	fbDiagnosisEtherCATSlaveWc0				:ARRAY[E_EtherCATSlave.Drive14_AZD4A_KED..E_EtherCATSlave.Drive14_AZD4A_KED] OF FB_DiagnosisEtherCATSlaveWc0
																														(	E_EtherCATSlave.Drive14_AZD4A_KED
																															);	//EtherCAT Slave診断用FB
END_VAR

bError:=EtherCATMasterDiagnosis() OR EtherCATSlaveDiagnosis();

METHOD INTERNAL EtherCATMasterDiagnosis : BOOL
//EtherCATマスター診断
	//デバイス2
	fbDiagnosisEtherCATMaster2(	fbFrmWcStateDiagnosis	:=fbFrmWcStateDiagnosis2,
								fbFrmStateDiagnosis		:=fbFrmStateDiagnosis2);

	//デバイス6
	fbDiagnosisEtherCATMaster6(	fbFrmWcStateDiagnosis	:=fbFrmWcStateDiagnosis6,
								fbFrmStateDiagnosis		:=fbFrmStateDiagnosis6);

	//すべて問題なしで出力
	EtherCATMasterDiagnosis:= fbDiagnosisEtherCATMaster2.bError OR fbDiagnosisEtherCATMaster6.bError;
END_METHOD

METHOD INTERNAL EtherCATSlaveDiagnosis : BOOL
//EtherCATスレーブ診断
	fbDiagnosisEtherCATSlaveWc2[E_EtherCATSlave.Term12_EL2911]();
	fbDiagnosisEtherCATSlaveWc0[E_EtherCATSlave.Drive14_AZD4A_KED]();
	
	EtherCATSlaveDiagnosis:=fbDiagnosisEtherCATSlaveWc2[E_EtherCATSlave.Term12_EL2911].bError OR fbDiagnosisEtherCATSlaveWc0[E_EtherCATSlave.Drive14_AZD4A_KED].bError;

	FOR eEtherCATSlave := E_EtherCATSlave.Term2_EL9410 TO E_EtherCATSlave.Term11_EL1088 DO
		fbDiagnosisEtherCATSlaveWc1[eEtherCATSlave]();
		EtherCATSlaveDiagnosis:=EtherCATSlaveDiagnosis OR fbDiagnosisEtherCATSlaveWc1[eEtherCATSlave].bError;
	END_FOR
END_METHOD

END_FUNCTION_BLOCK

// ---- 01_Submodules/Diagnosis/EtherCAT Master/FB_FrmWcStateDiagnosis.TcPOU
FUNCTION_BLOCK FB_FrmWcStateDiagnosis
VAR_IN_OUT
	eEtherCATMaster				:E_EtherCATMaster;	
END_VAR
VAR_OUTPUT
	bError						:BOOL;								//エラー発生を出力
END_VAR
VAR
	uiFrmWcState 		AT%I*	:UINT;								//PDデータとリンク
	
	sMasterName					:STRING;
	
	bErrorState					:ARRAY[0..15] OF BOOL;				//各ステートエラー
	fbBitREdge					:ARRAY[0..15] OF R_TRIG;
	bSendMsgMem					:ARRAY[0..14] OF BOOL;				//メッセージ送信を記憶	
	sSendMsgString				:STRING;							//送信メッセージのアーギュメント用
	bSendMsg					:BOOL;								//メッセージ送信予約
	fbMessage					:ARRAY[0..1] OF FB_TcMessage;
	i							:INT;
END_VAR

//マスター名を入力
	IF sMasterName<>TO_STRING(eEtherCATMaster) THEN
		sMasterName:=TO_STRING(eEtherCATMaster);
	END_IF

//エラー状態を出力
	bError:= uiFrmWcState<>0 ;
	
//サイクリックフレームごとのワーキングカウンターチェック、エラーは複数発生する可能性があるので全bitチェック
	FOR i := 0 TO 15 DO
		bErrorState[i]:=(uiFrmWcState AND SHL(1,i))<>0;
	END_FOR
	
//結果をEventloggerへ
	bSendMsg:=FALSE;	//メッセージ送信予約をリセット

	FOR i := 0 TO 14 BY 1 DO
		//エラーの立ち上がりエッジを検出
		fbBitREdge[i](CLK:=bErrorState[i]);
		
		//まだ送信していなければ、送信用の文字列作成
		IF NOT bSendMsgMem[i] AND fbBitREdge[i].Q THEN
			
			sSendMsgString:=CONCAT(sSendMsgString, CONCAT(INT_TO_STRING(i+1), '. '));	//送信メッセージのアーギュメント作成

			bSendMsg:=TRUE;		//メッセージ送信予約をセット
			bSendMsgMem[i]:=TRUE;	//メッセージ送信を記憶
			
		END_IF
		
		//エラーがリセットされたらメッセージ送信気を記憶をリセット
		IF NOT bErrorState[i] THEN
			bSendMsgMem[i]:=FALSE;
		END_IF
		
	END_FOR
	
	IF bSendMsg THEN
		fbMessage[0].ipArguments.Clear().AddString(sSendMsgString).AddString(sMasterName);
		fbMessage[0].Send();
		
		bSendMsg:=FALSE;
		sSendMsgString:='';
	END_IF
	
	//全体判定用
	fbBitREdge[15](CLK:=bErrorState[15]);
	
	IF fbBitREdge[15].Q THEN
		fbMessage[1].ipArguments.Clear().AddString(sMasterName);
		fbMessage[1].Send();
	END_IF

//FB_Init は常に暗黙的に使用可能で、主に初期化に使用されます。
//戻り値は評価されません。特定の結果を得るために、メソッドを明示的に宣言し、
//そのメソッドに標準の初期化コードをもったコードを追加することができます。戻り値を評価できます。
METHOD FB_Init: BOOL
VAR_INPUT
    bInitRetains: BOOL; // TRUE: 保持変数は初期化されます (ウォーム リセット、あるいはコールド リセット)
    bInCopyCode: BOOL;  // TRUE: 後でコードをコピーする (オンライン変更) ために、インスタンスをコピーします。
END_VAR
fbMessage[0].CreateEx(TC_EVENTS.TkEtherCATMasterDiagnosisEventClass.WrongWorkingCounterEtherCATCommandReceived);
fbMessage[1].CreateEx(TC_EVENTS.TkEtherCATMasterDiagnosisEventClass.CompleteFrameMissing);
END_METHOD

END_FUNCTION_BLOCK

// ---- 01_Submodules/Diagnosis/EtherCAT Master/FB_FrmStateDiagnosis.TcPOU
FUNCTION_BLOCK FB_FrmStateDiagnosis
VAR_IN_OUT
	eEtherCATMaster				:E_EtherCATMaster;	
END_VAR
VAR_OUTPUT
	bError						:BOOL;								//エラー発生を出力
END_VAR
VAR
	uiFrmState 			AT%I*	:UINT;								//PDデータとリンク
	
	sMasterName					:STRING;
	
	bErrorState					:ARRAY[0..15] OF BOOL;				//各ステートエラー
	fbBitREdge					:ARRAY[0..15] OF R_TRIG;
	bSendMsgMem					:ARRAY[0..14] OF BOOL;				//メッセージ送信を記憶	
	sSendMsgString				:STRING;							//送信メッセージのアーギュメント用
	bSendMsg					:BOOL;								//メッセージ送信予約
	fbMessage					:ARRAY[0..1] OF FB_TcMessage;
	i							:INT;
END_VAR

//マスター名を入力
	IF sMasterName<>TO_STRING(eEtherCATMaster) THEN
		sMasterName:=TO_STRING(eEtherCATMaster);
	END_IF

//エラー状態を出力
	bError:= uiFrmState<>0 ;
	
//サイクリックフレームごとのワーキングカウンターチェック、エラーは複数発生する可能性があるので全bitチェック
	FOR i := 0 TO 15 DO
		bErrorState[i]:=(uiFrmState AND SHL(1,i))<>0;
	END_FOR
	
//結果をEventloggerへ
	bSendMsg:=FALSE;	//メッセージ送信予約をリセット

	FOR i := 0 TO 14 BY 1 DO
		//エラーの立ち上がりエッジを検出
		fbBitREdge[i](CLK:=bErrorState[i]);
		
		//まだ送信していなければ、送信用の文字列作成
		IF NOT bSendMsgMem[i] AND fbBitREdge[i].Q THEN
			
			sSendMsgString:=CONCAT(sSendMsgString, CONCAT(INT_TO_STRING(i+1), '. '));	//送信メッセージのアーギュメント作成

			bSendMsg:=TRUE;		//メッセージ送信予約をセット
			bSendMsgMem[i]:=TRUE;	//メッセージ送信を記憶
			
		END_IF
		
		//エラーがリセットされたらメッセージ送信気を記憶をリセット
		IF NOT bErrorState[i] THEN
			bSendMsgMem[i]:=FALSE;
		END_IF
		
	END_FOR
	
	IF bSendMsg THEN
		fbMessage[0].ipArguments.Clear().AddString(sSendMsgString).AddString(sMasterName);
		fbMessage[0].Send();
		
		bSendMsg:=FALSE;
		sSendMsgString:='';
	END_IF
	
	//全体判定用
	fbBitREdge[15](CLK:=bErrorState[15]);
	
	IF fbBitREdge[15].Q THEN
		fbMessage[1].ipArguments.Clear().AddString(sMasterName);
		fbMessage[1].Send();
	END_IF

//FB_Init は常に暗黙的に使用可能で、主に初期化に使用されます。
//戻り値は評価されません。特定の結果を得るために、メソッドを明示的に宣言し、
//そのメソッドに標準の初期化コードをもったコードを追加することができます。戻り値を評価できます。
METHOD FB_Init: BOOL
VAR_INPUT
    bInitRetains: BOOL; // TRUE: 保持変数は初期化されます (ウォーム リセット、あるいはコールド リセット)
    bInCopyCode: BOOL;  // TRUE: 後でコードをコピーする (オンライン変更) ために、インスタンスをコピーします。
END_VAR
fbMessage[0].CreateEx(TC_EVENTS.TkEtherCATMasterDiagnosisEventClass.EtherCATCommandNotSentNOPRequested);
fbMessage[1].CreateEx(TC_EVENTS.TkEtherCATMasterDiagnosisEventClass.CompleteFrameNotSent);
END_METHOD

END_FUNCTION_BLOCK

// ---- 01_Submodules/Diagnosis/EtherCAT Master/FB_DiagnosisEtherCATMaster.TcPOU
FUNCTION_BLOCK FB_DiagnosisEtherCATMaster
VAR_OUTPUT
	bError						:BOOL;								//エラー発生を出力
END_VAR
VAR_IN_OUT
	fbFrmWcStateDiagnosis		:ARRAY[*] OF FB_FrmWcStateDiagnosis;
	fbFrmStateDiagnosis			:ARRAY[*] OF FB_FrmStateDiagnosis;
END_VAR
VAR
	_eEtherCATMaster			:E_EtherCATMaster;	

	fbDevStateDiagnosis			:FB_DevStateDiagnosis;
	fbSlaveCountDiagnosis		:FB_SlaveCountDiagnosis;
	i							:DINT;
END_VAR

//診断用FBを呼び出し
fbDevStateDiagnosis(eEtherCATMaster:=_eEtherCATMaster);
fbSlaveCountDiagnosis(eEtherCATMaster:=_eEtherCATMaster);

bError:=fbDevStateDiagnosis.bError OR fbSlaveCountDiagnosis.bError;

//可変長のアレイを診断と出力
FOR i := LOWER_BOUND(fbFrmWcStateDiagnosis,1) TO UPPER_BOUND(fbFrmWcStateDiagnosis,1) DO
	fbFrmWcStateDiagnosis[i](eEtherCATMaster:=_eEtherCATMaster);
	bError:=bError OR fbFrmWcStateDiagnosis[i].bError;
END_FOR

FOR i := LOWER_BOUND(fbFrmStateDiagnosis,1) TO UPPER_BOUND(fbFrmStateDiagnosis,1) DO
	fbFrmStateDiagnosis[i](eEtherCATMaster:=_eEtherCATMaster);
	bError:=bError OR fbFrmStateDiagnosis[i].bError;
END_FOR

//FB_Init は常に暗黙的に使用可能で、主に初期化に使用されます。
//戻り値は評価されません。特定の結果を得るために、メソッドを明示的に宣言し、
//そのメソッドに標準の初期化コードをもったコードを追加することができます。戻り値を評価できます。
METHOD FB_Init: BOOL
VAR_INPUT
    bInitRetains: BOOL; // TRUE: 保持変数は初期化されます (ウォーム リセット、あるいはコールド リセット)
    bInCopyCode: BOOL;  // TRUE: 後でコードをコピーする (オンライン変更) ために、インスタンスをコピーします。
	
	eEtherCATMaster	:E_EtherCATMaster;
END_VAR
_eEtherCATMaster:=eEtherCATMaster;
END_METHOD

END_FUNCTION_BLOCK

// ---- 01_Submodules/Diagnosis/EtherCAT Master/FB_DevStateDiagnosis.TcPOU
FUNCTION_BLOCK FB_DevStateDiagnosis
VAR CONSTANT
	uiFaultMask					:UINT	:=2#0001_1111_1111_0011;	//デバイスエラーのマスク
END_VAR
VAR_IN_OUT
	eEtherCATMaster				:E_EtherCATMaster;	
END_VAR
VAR_OUTPUT
	bError						:BOOL;								//エラー発生を出力
END_VAR
VAR
	uiDevState 			AT%I*	:UINT;								//PDデータとリンク
	
	sMasterName					:STRING;
	
	bErrorState					:ARRAY[0..15] OF BOOL;				//各ステートエラー
	fbBitREdge					:ARRAY[0..15] OF R_TRIG;
	fbMessage					:ARRAY[0..15] OF FB_TcMessage;
	i							:INT;
END_VAR

//マスター名を入力
	IF sMasterName<>TO_STRING(eEtherCATMaster) THEN
		sMasterName:=TO_STRING(eEtherCATMaster);
	END_IF

//エラー状態を出力
	bError:= (uiDevState AND uiFaultMask)<>0 ;

//デバイスの状態チェック、エラーは複数発生する可能性があるので全bitチェック
	FOR i := 0 TO 15 DO
		bErrorState[i]:=(uiDevState AND SHL(1,i))<>0;
	END_FOR

//結果をEventloggerへ
	FOR i := 0 TO 15 BY 1 DO
		fbBitREdge[i](CLK:=bErrorState[i]);
		
		IF fbBitREdge[i].Q THEN
			fbMessage[i].ipArguments.Clear().AddString(sMasterName);
			fbMessage[i].Send();
		END_IF
		
	END_FOR

//FB_Init は常に暗黙的に使用可能で、主に初期化に使用されます。
//戻り値は評価されません。特定の結果を得るために、メソッドを明示的に宣言し、
//そのメソッドに標準の初期化コードをもったコードを追加することができます。戻り値を評価できます。
METHOD FB_Init: BOOL
VAR_INPUT
    bInitRetains: BOOL; // TRUE: 保持変数は初期化されます (ウォーム リセット、あるいはコールド リセット)
    bInCopyCode: BOOL;  // TRUE: 後でコードをコピーする (オンライン変更) ために、インスタンスをコピーします。
END_VAR
fbMessage[0].CreateEx(TC_EVENTS.TkEtherCATMasterDiagnosisEventClass.LinkError);
fbMessage[1].CreateEx(TC_EVENTS.TkEtherCATMasterDiagnosisEventClass.IOLockedAfterLinkErrorIOResetRequired);
fbMessage[2].CreateEx(TC_EVENTS.TkEtherCATMasterDiagnosisEventClass.LinkErrorRedundancyAdapter);
fbMessage[3].CreateEx(TC_EVENTS.TkEtherCATMasterDiagnosisEventClass.MissingOneFrameRedundancyAdapter);
fbMessage[4].CreateEx(TC_EVENTS.TkEtherCATMasterDiagnosisEventClass.OutOfSendResourcesIOResetRequired);
fbMessage[5].CreateEx(TC_EVENTS.TkEtherCATMasterDiagnosisEventClass.WatchdogTriggered);
fbMessage[6].CreateEx(TC_EVENTS.TkEtherCATMasterDiagnosisEventClass.EthernetDriverMiniportNotFound);
fbMessage[7].CreateEx(TC_EVENTS.TkEtherCATMasterDiagnosisEventClass.IOResetActive);
fbMessage[8].CreateEx(TC_EVENTS.TkEtherCATMasterDiagnosisEventClass.AtLeastOneDeviceInINITState);
fbMessage[9].CreateEx(TC_EVENTS.TkEtherCATMasterDiagnosisEventClass.AtLeastOneDeviceInPREOPState);
fbMessage[10].CreateEx(TC_EVENTS.TkEtherCATMasterDiagnosisEventClass.AtLeastOneDeviceInSAFEOPState);
fbMessage[11].CreateEx(TC_EVENTS.TkEtherCATMasterDiagnosisEventClass.AtLeastOneDeviceInERRORState);
fbMessage[12].CreateEx(TC_EVENTS.TkEtherCATMasterDiagnosisEventClass.DCNotInSync);
END_METHOD

END_FUNCTION_BLOCK

// ---- 01_Submodules/Diagnosis/EtherCAT Master/FB_SlaveCountDiagnosis.TcPOU
FUNCTION_BLOCK FB_SlaveCountDiagnosis
VAR_IN_OUT
	eEtherCATMaster				:E_EtherCATMaster;	
END_VAR
VAR_OUTPUT
	bError						:BOOL;								//エラー発生を出力
END_VAR
VAR
	uiSlaveCount 		AT%I*	:UINT;								//PDデータとリンク
	uiCfgSlaveCount 	AT%I*	:UINT;								//PDデータとリンク
	
	sMasterName					:STRING;
	
	fbBitREdge					:R_TRIG;
	fbMessage					:FB_TcMessage;
	i							:INT;
END_VAR

//マスター名を入力
	IF sMasterName<>TO_STRING(eEtherCATMaster) THEN
		sMasterName:=TO_STRING(eEtherCATMaster);
	END_IF

//エラー状態を出力
	bError:=uiSlaveCount<>uiCfgSlaveCount OR uiSlaveCount=0 OR uiCfgSlaveCount=0;

//エラーをEventloggerへ
	fbBitREdge(CLK:=bError);
	
	IF fbBitREdge.Q THEN
		fbMessage.ipArguments.Clear().AddString(sMasterName);
		fbMessage.Send();
	END_IF

//FB_Init は常に暗黙的に使用可能で、主に初期化に使用されます。
//戻り値は評価されません。特定の結果を得るために、メソッドを明示的に宣言し、
//そのメソッドに標準の初期化コードをもったコードを追加することができます。戻り値を評価できます。
METHOD FB_Init: BOOL
VAR_INPUT
    bInitRetains: BOOL; // TRUE: 保持変数は初期化されます (ウォーム リセット、あるいはコールド リセット)
    bInCopyCode: BOOL;  // TRUE: 後でコードをコピーする (オンライン変更) ために、インスタンスをコピーします。
END_VAR
fbMessage.CreateEx(Tc_Events.TkEtherCATMasterDiagnosisEventClass.MismatchSlaveCountCfgSlaveCount);
END_METHOD

END_FUNCTION_BLOCK

// ---- 01_Submodules/Diagnosis/EtherCAT Slave/FB_DiagnosisEtherCATSlaveWc1.TcPOU
FUNCTION_BLOCK FB_DiagnosisEtherCATSlaveWc1
VAR_OUTPUT
	bError						:BOOL;								//エラー発生を出力
END_VAR
VAR
	_eEtherCATSlave				:E_EtherCATSlave;
	
	fbStateDiagnosis			:FB_StateDiagnosis;
	fbWcStateDiagnosis			:FB_WcStateDiagnosis;
END_VAR

//診断用FBを呼び出し
fbStateDiagnosis(eEtherCATSlave:=_eEtherCATSlave);
fbWcStateDiagnosis(eEtherCATSlave:=_eEtherCATSlave);

bError:=fbStateDiagnosis.bError OR fbWcStateDiagnosis.bError;

//FB_Init は常に暗黙的に使用可能で、主に初期化に使用されます。
//戻り値は評価されません。特定の結果を得るために、メソッドを明示的に宣言し、
//そのメソッドに標準の初期化コードをもったコードを追加することができます。戻り値を評価できます。
METHOD FB_Init: BOOL
VAR_INPUT
    bInitRetains: BOOL; // TRUE: 保持変数は初期化されます (ウォーム リセット、あるいはコールド リセット)
    bInCopyCode: BOOL;  // TRUE: 後でコードをコピーする (オンライン変更) ために、インスタンスをコピーします。

	eEtherCATSlave							:E_EtherCATSlave;
END_VAR
_eEtherCATSlave:=eEtherCATSlave;
END_METHOD

END_FUNCTION_BLOCK

// ---- 01_Submodules/Diagnosis/EtherCAT Slave/FB_StateDiagnosis.TcPOU
FUNCTION_BLOCK FB_StateDiagnosis
VAR CONSTANT
	uiFaultMask					:UINT	:=2#1111_1111_1111_0111;	//デバイスエラーのマスク
END_VAR
VAR_IN_OUT
	eEtherCATSlave				:E_EtherCATSlave;
END_VAR
VAR_OUTPUT
	bError						:BOOL;								//エラー発生を出力
END_VAR
VAR
	uiState				AT%I*	:UINT;								//PDデータとリンク
	
	sSlaveName					:STRING;
	
	bErrorState					:ARRAY[0..16] OF BOOL;				//各ステートエラー
	fbBitREdge					:ARRAY[0..16] OF R_TRIG;
	fbMessage					:ARRAY[0..16] OF FB_TcMessage;
	i							:INT;
END_VAR

//スレーブ名を入力
	IF sSlaveName<>TO_STRING(eEtherCATSlave) THEN
		sSlaveName:=TO_STRING(eEtherCATSlave);
	END_IF

//エラー状態を出力
	bError:= (uiState AND uiFaultMask)<>0 ;

//スレーブのステータスをbitから診断
	bErrorState[0]:=uiState.0 AND NOT uiState.1;
	bErrorState[1]:=uiState.1 AND NOT uiState.0;
	bErrorState[2]:=uiState.0 AND uiState.1;
	bErrorState[3]:=uiState.2;
	bErrorState[4]:=uiState.3;

//スレーブのエラーは複数発生する可能性があるので全bitチェック
	FOR i := 4 TO 15 DO
		bErrorState[i+1]:=(uiState AND SHL(1,i))<>0;
	END_FOR

//結果をEventloggerへ
	FOR i := 0 TO 16 BY 1 DO
		fbBitREdge[i](CLK:=bErrorState[i]);
		
		IF fbBitREdge[i].Q THEN
			fbMessage[i].ipArguments.Clear().AddString(sSlaveName);
			fbMessage[i].Send();
		END_IF
		
	END_FOR

//FB_Init は常に暗黙的に使用可能で、主に初期化に使用されます。
//戻り値は評価されません。特定の結果を得るために、メソッドを明示的に宣言し、
//そのメソッドに標準の初期化コードをもったコードを追加することができます。戻り値を評価できます。
METHOD FB_Init: BOOL
VAR_INPUT
    bInitRetains: BOOL; // TRUE: 保持変数は初期化されます (ウォーム リセット、あるいはコールド リセット)
    bInCopyCode: BOOL;  // TRUE: 後でコードをコピーする (オンライン変更) ために、インスタンスをコピーします。
END_VAR
fbMessage[0].CreateEx(TC_EVENTS.TkEtherCATSlaveDiagnosisEventClass.INIT);
fbMessage[1].CreateEx(TC_EVENTS.TkEtherCATSlaveDiagnosisEventClass.PREOP);
fbMessage[2].CreateEx(TC_EVENTS.TkEtherCATSlaveDiagnosisEventClass.BOOT);
fbMessage[3].CreateEx(TC_EVENTS.TkEtherCATSlaveDiagnosisEventClass.SAFEOP);
fbMessage[4].CreateEx(TC_EVENTS.TkEtherCATSlaveDiagnosisEventClass.OP);
fbMessage[5].CreateEx(TC_EVENTS.TkEtherCATSlaveDiagnosisEventClass.SlaveSignalsError);
fbMessage[6].CreateEx(TC_EVENTS.TkEtherCATSlaveDiagnosisEventClass.InvalidVendorIdProductCodeRead);
fbMessage[7].CreateEx(TC_EVENTS.TkEtherCATSlaveDiagnosisEventClass.InitializationErrorOccurred);
fbMessage[8].CreateEx(TC_EVENTS.TkEtherCATSlaveDiagnosisEventClass.SlaveDisabled);
fbMessage[9].CreateEx(TC_EVENTS.TkEtherCATSlaveDiagnosisEventClass.SlaveNotPresent);
fbMessage[10].CreateEx(TC_EVENTS.TkEtherCATSlaveDiagnosisEventClass.SlaveSignalsLinkError);
fbMessage[11].CreateEx(TC_EVENTS.TkEtherCATSlaveDiagnosisEventClass.SlaveSignalsMissingLink);
fbMessage[12].CreateEx(TC_EVENTS.TkEtherCATSlaveDiagnosisEventClass.SlaveSlaveSignalsUnexpectedLink);
fbMessage[13].CreateEx(TC_EVENTS.TkEtherCATSlaveDiagnosisEventClass.CommunicationPortA);
fbMessage[14].CreateEx(TC_EVENTS.TkEtherCATSlaveDiagnosisEventClass.CommunicationPortB);
fbMessage[15].CreateEx(TC_EVENTS.TkEtherCATSlaveDiagnosisEventClass.CommunicationPortC);
fbMessage[16].CreateEx(TC_EVENTS.TkEtherCATSlaveDiagnosisEventClass.CommunicationPortD);
END_METHOD

END_FUNCTION_BLOCK

// ---- 01_Submodules/Diagnosis/EtherCAT Slave/FB_WcStateDiagnosis.TcPOU
FUNCTION_BLOCK FB_WcStateDiagnosis
VAR_IN_OUT
	eEtherCATSlave				:E_EtherCATSlave;
END_VAR
VAR_OUTPUT
	bError						:BOOL;								//エラー発生を出力
END_VAR
VAR
	bWcState			AT%I*	:BOOL;								//PDデータとリンク
	
	sSlaveName					:STRING;
	
	fbBitREdge					:R_TRIG;
	fbMessage					:FB_TcMessage;
END_VAR

//スレーブ名を入力
	IF sSlaveName<>TO_STRING(eEtherCATSlave) THEN
		sSlaveName:=TO_STRING(eEtherCATSlave);
	END_IF

//エラー状態を出力
	bError:=bWcState;

//結果をEventloggerへ
	fbBitREdge(CLK:=bError);
	
	IF fbBitREdge.Q THEN
		fbMessage.ipArguments.Clear().AddString(sSlaveName);
		fbMessage.Send();
	END_IF

//FB_Init は常に暗黙的に使用可能で、主に初期化に使用されます。
//戻り値は評価されません。特定の結果を得るために、メソッドを明示的に宣言し、
//そのメソッドに標準の初期化コードをもったコードを追加することができます。戻り値を評価できます。
METHOD FB_Init: BOOL
VAR_INPUT
    bInitRetains: BOOL; // TRUE: 保持変数は初期化されます (ウォーム リセット、あるいはコールド リセット)
    bInCopyCode: BOOL;  // TRUE: 後でコードをコピーする (オンライン変更) ために、インスタンスをコピーします。
END_VAR
fbMessage.CreateEx(TC_EVENTS.TkEtherCATSlaveDiagnosisEventClass.InvalidWorkingCounter);
END_METHOD

END_FUNCTION_BLOCK

// ---- 01_Submodules/Diagnosis/EtherCAT Slave/FB_DiagnosisEtherCATSlaveWc2.TcPOU
FUNCTION_BLOCK FB_DiagnosisEtherCATSlaveWc2
VAR_OUTPUT
	bError						:BOOL;								//エラー発生を出力
END_VAR
VAR
	_eEtherCATSlave				:E_EtherCATSlave;
	
	fbStateDiagnosis			:FB_StateDiagnosis;
	fbWcStateDiagnosis1			:FB_WcStateDiagnosis;
	fbWcStateDiagnosis2			:FB_WcStateDiagnosis;
END_VAR

//診断用FBを呼び出し
fbStateDiagnosis(eEtherCATSlave:=_eEtherCATSlave);
fbWcStateDiagnosis1(eEtherCATSlave:=_eEtherCATSlave);
fbWcStateDiagnosis2(eEtherCATSlave:=_eEtherCATSlave);

bError:=fbStateDiagnosis.bError OR fbWcStateDiagnosis1.bError OR fbWcStateDiagnosis2.bError;

//FB_Init は常に暗黙的に使用可能で、主に初期化に使用されます。
//戻り値は評価されません。特定の結果を得るために、メソッドを明示的に宣言し、
//そのメソッドに標準の初期化コードをもったコードを追加することができます。戻り値を評価できます。
METHOD FB_Init: BOOL
VAR_INPUT
    bInitRetains: BOOL; // TRUE: 保持変数は初期化されます (ウォーム リセット、あるいはコールド リセット)
    bInCopyCode: BOOL;  // TRUE: 後でコードをコピーする (オンライン変更) ために、インスタンスをコピーします。

	eEtherCATSlave							:E_EtherCATSlave;
END_VAR
_eEtherCATSlave:=eEtherCATSlave;
END_METHOD

END_FUNCTION_BLOCK

// ---- 01_Submodules/Diagnosis/EtherCAT Slave/FB_DiagnosisEtherCATSlaveWc0.TcPOU
FUNCTION_BLOCK FB_DiagnosisEtherCATSlaveWc0
VAR_OUTPUT
	bError						:BOOL;								//エラー発生を出力
END_VAR
VAR
	_eEtherCATSlave				:E_EtherCATSlave;
	
	fbStateDiagnosis			:FB_StateDiagnosis;
END_VAR

//診断用FBを呼び出し
fbStateDiagnosis(eEtherCATSlave:=_eEtherCATSlave);

bError:=fbStateDiagnosis.bError;

//FB_Init は常に暗黙的に使用可能で、主に初期化に使用されます。
//戻り値は評価されません。特定の結果を得るために、メソッドを明示的に宣言し、
//そのメソッドに標準の初期化コードをもったコードを追加することができます。戻り値を評価できます。
METHOD FB_Init: BOOL
VAR_INPUT
    bInitRetains: BOOL; // TRUE: 保持変数は初期化されます (ウォーム リセット、あるいはコールド リセット)
    bInCopyCode: BOOL;  // TRUE: 後でコードをコピーする (オンライン変更) ために、インスタンスをコピーします。

	eEtherCATSlave							:E_EtherCATSlave;
END_VAR
_eEtherCATSlave:=eEtherCATSlave;
END_METHOD

END_FUNCTION_BLOCK

// ---- 01_Submodules/MachineState/FB_MachineState.TcPOU
FUNCTION_BLOCK FB_MachineState EXTENDS FB_ListenerBase2
VAR_INPUT
	bCritical					:BOOL;				//クリティカルの発生
	bError						:BOOL;				//エラーの発生
	bWarning					:BOOL;				//ワーニングの発生
	bStay						:BOOL;				//McPowerがOFF
	bStop						:BOOL;				//McPowerがON
	bMoving						:BOOL;				//軸動作中または、（自動動作実行中（まだない））
END_VAR
VAR_OUTPUT
	eMachineState				:E_MachineState;	//マシーンステートを出力
	bStopMachine				:BOOL;				//モーションファンクションブロック停止
END_VAR
VAR
	fbListenerFilter			:FB_TcEventFilter;	//アラームフィルター

	liCriticalActiveCount		:LINT;				//クリティカル発生状況記憶
	liErrorActiveCount			:LINT;				//エラー発生状況記憶
	liWarningActiveCount		:LINT;				//ワーニング発生状況記憶
END_VAR

//---常に呼び出す必要があるので呼び出し---
	SUPER^.Execute();

//---発生アラームの重いほうからマシンステートに登録---
	IF bCritical=TRUE OR liCriticalActiveCount<>0 THEN
		eMachineState:=E_MachineState.Critical;
		bStopMachine:=TRUE;
		
	ELSIF bError=TRUE OR liErrorActiveCount<>0 THEN
		eMachineState:=E_MachineState.Error;
		bStopMachine:=TRUE;
	
	ELSIF bWarning=TRUE OR liWarningActiveCount<>0 THEN
		eMachineState:=E_MachineState.Warning;
		bStopMachine:=FALSE;
		
	ELSIF bStay=TRUE THEN
		eMachineState:=E_MachineState.Stay;
		bStopMachine:=FALSE;
		
	ELSIF bStop=TRUE THEN
		eMachineState:=E_MachineState.Stop;
		bStopMachine:=FALSE;
		
	ELSIF bMoving=TRUE THEN
		eMachineState:=E_MachineState.Moving;
		bStopMachine:=FALSE;
	END_IF

//FB_Init は常に暗黙的に使用可能で、主に初期化に使用されます。
//戻り値は評価されません。特定の結果を得るために、メソッドを明示的に宣言し、
//そのメソッドに標準の初期化コードをもったコードを追加することができます。戻り値を評価できます。
METHOD FB_Init: BOOL
VAR_INPUT
    bInitRetains: BOOL; // TRUE: 保持変数は初期化されます (ウォーム リセット、あるいはコールド リセット)
    bInCopyCode: BOOL;  // TRUE: 後でコードをコピーする (オンライン変更) ために、インスタンスをコピーします。
END_VAR
IF bInCopyCode = FALSE THEN
	
	//継承元のファンクションブロックの読み込むイベントのフィルター設定、アラームをフィルタリング
	fbListenerFilter.Clear().IsAlarm();
	
	//設定したフィルターを設定する
	SUPER^.Subscribe2(fbListenerFilter);

END_IF
END_METHOD

METHOD OnAlarmCleared : Tc3_EventLogger.HRESULT
VAR_INPUT
	fbEvent	: REFERENCE TO Tc3_EventLogger.FB_TcEvent;
END_VAR
CASE fbEvent.eSeverity OF 
	TcEventSeverity.Critical:
		liCriticalActiveCount:=liCriticalActiveCount-1;
		
	TcEventSeverity.Error:
		liErrorActiveCount:=liErrorActiveCount-1;
		
	TcEventSeverity.Warning:
		liWarningActiveCount:=liWarningActiveCount-1;
END_CASE

OnAlarmCleared:=S_OK;
END_METHOD

METHOD OnAlarmRaised : Tc3_EventLogger.HRESULT
VAR_INPUT
	fbEvent	: REFERENCE TO Tc3_EventLogger.FB_TcEvent;
END_VAR
CASE fbEvent.eSeverity OF 
	TcEventSeverity.Critical:
		liCriticalActiveCount:=liCriticalActiveCount+1;
		
	TcEventSeverity.Error:
		liErrorActiveCount:=liErrorActiveCount+1;
		
	TcEventSeverity.Warning:
		liWarningActiveCount:=liWarningActiveCount+1;
END_CASE

OnAlarmRaised:=S_OK;
END_METHOD

END_FUNCTION_BLOCK

// ---- 01_Submodules/Alarm/FB_Alarm.TcPOU
FUNCTION_BLOCK FB_Alarm EXTENDS FB_TcAlarm
VAR_INPUT
	bRaise				:BOOL;				//アラーム発生
	bClear				:BOOL;				//アラームクリア
	bConfirm			:BOOL;				//アラーム確認
END_VAR
VAR_OUTPUT
END_VAR
VAR
	h					:HRESULT;
	hError				:HRESULT;
	
	REdge				:R_TRIG;			//アラーム発生の立ち上がりエッジ
	bRaiseMem			:BOOL;				//アラーム発生を保持
END_VAR

//アラーム発生の立ち上がりエッジ検出
REdge(CLK := bRaise);

IF REdge.Q AND (NOT SUPER^.bRaised) THEN
	bRaiseMem	:=TRUE;
END_IF

//Raise
IF bRaiseMem AND (NOT SUPER^.bRaised) THEN
	h:=SUPER^.Raise(0);
	IF FAILED(h) THEN
		hError := h;
	END_IF
	bRaiseMem:=FALSE;
END_IF

//Confirm
IF bConfirm AND SUPER^.eConfirmationState=TCEVENTCONFIRMATIONSTATE.WaitForConfirmation THEN
	h:=SUPER^.Confirm(0);
	IF FAILED(h) THEN
		hError := h;
	END_IF
END_IF

//Clear
IF (NOT bRaise) AND bClear AND SUPER^.bRaised THEN
	h:=SUPER^.Clear(0 ,FALSE);
	IF FAILED(h) THEN
		hError := h;
	END_IF
END_IF

METHOD FB_init : BOOL
VAR_INPUT
	bInitRetains 	: BOOL; // if TRUE, the retain variables are initialized (warm start / cold start)
	bInCopyCode 	: BOOL;  // if TRUE, the instance afterwards gets moved into the copy code (online change)
	TcEvtEntry		:TcEventEntry;
END_VAR
SUPER^.CreateEx(TcEvtEntry, TRUE, 0);
END_METHOD

END_FUNCTION_BLOCK

// ---- 01_Submodules/Alarm/FB_AlarmFromTcMessage.TcPOU
FUNCTION_BLOCK FB_AlarmFromTcMessage EXTENDS FB_TcAlarm
VAR_INPUT
	bRaise				:BOOL;				//アラーム発生
	bClear				:BOOL;				//アラームクリア
	bConfirm			:BOOL;				//アラーム確認
	ipResultMessage		:I_TcMessage;		//アラームメッセージ(I_TcMessage)
END_VAR
VAR_OUTPUT
END_VAR
VAR
	h					:HRESULT;
	hError				:HRESULT;
	
	REdge				:R_TRIG;			//アラーム発生の立ち上がりエッジ
	bRaiseMem			:BOOL;				//アラーム発生を保持
	bLinked				:BOOL;				//アラームメッセージのCreateEx済みフラグ
END_VAR

//アラーム発生の立ち上がりエッジ検出
REdge(CLK := bRaise);

IF REdge.Q AND (NOT SUPER^.bRaised) THEN
	bRaiseMem	:=TRUE;
	bLinked		:=FALSE;
END_IF
 
//CreateEx
IF bRaiseMem AND (NOT bLinked) AND (ipResultMessage <> 0) THEN
	SUPER^.CreateEx(stEventEntry:=ipResultMessage.stEventEntry,	TRUE, ipSourceInfo := ipResultMessage.ipSourceInfo);
	bLinked:=TRUE;
END_IF
 
//Raise
IF bRaiseMem AND bLinked AND (NOT SUPER^.bRaised) THEN
	h:=SUPER^.Raise(0);
	IF FAILED(h) THEN
		hError := h;
	END_IF
	bRaiseMem:=FALSE;
END_IF
 
//Confirm
IF bConfirm AND (SUPER^.eConfirmationState = TCEVENTCONFIRMATIONSTATE.WaitForConfirmation) THEN
	h:=SUPER^.Confirm(0);
	IF FAILED(h) THEN
		hError := h;
	END_IF
END_IF
 
//Clear
IF (NOT bRaise) AND bClear AND SUPER^.bRaised THEN
	h:=SUPER^.Clear(0 ,FALSE);
	IF FAILED(h) THEN
		hError := h;
	END_IF
END_IF

END_FUNCTION_BLOCK

// ---- 01_Submodules/FB_PersistentDataManagement.TcPOU
FUNCTION_BLOCK FB_PersistentDataManagement
VAR
	fbWritePersistentData		:FB_WritePersistentData;
	fbWriteREdge				:R_TRIG;
	fbWriteErrorREdge			:R_TRIG;
	PcAmsNetId					:AMSNETID;					//PC AMS Net ID
END_VAR
VAR PERSISTENT
	_bPersistentDataNotInit		:BOOL	:=FALSE;
END_VAR

PROPERTY bPersistentDataNotInit : BOOL
GET
bPersistentDataNotInit:=_bPersistentDataNotInit;
END_GET
SET
IF _bPersistentDataNotInit<>bPersistentDataNotInit THEN
	_bPersistentDataNotInit:=bPersistentDataNotInit;
	WritePersistentData(TRUE);
END_IF
END_SET
END_PROPERTY

//FB_Init は常に暗黙的に使用可能で、主に初期化に使用されます。
//戻り値は評価されません。特定の結果を得るために、メソッドを明示的に宣言し、
//そのメソッドに標準の初期化コードをもったコードを追加することができます。戻り値を評価できます。
METHOD FB_Init: BOOL
VAR_INPUT
    bInitRetains: BOOL; // TRUE: 保持変数は初期化されます (ウォーム リセット、あるいはコールド リセット)
    bInCopyCode: BOOL;  // TRUE: 後でコードをコピーする (オンライン変更) ために、インスタンスをコピーします。

	PcAmsNetId			:AMSNETID;		//PC AMS Net ID
END_VAR
THIS^.PcAmsNetId		:=PcAmsNetId;
END_METHOD

METHOD WritePersistentData : BOOL
VAR_INPUT
	bPersistentDataWrite		:BOOL;
END_VAR
	fbWriteREdge(CLK:=bPersistentDataWrite,Q=>);

	IF fbWriteREdge.Q=TRUE THEN
		fbWritePersistentData(	NETID	:=F_CreateAmsNetId(PcAmsNetId),
								PORT	:=_AppInfo.AdsPort,
								START	:=TRUE,
								TMOUT	:=DEFAULT_ADS_TIMEOUT,
								MODE	:=E_PersistentMode.SPDM_2PASS,
								BUSY	=>,
								ERR		=>,
								ERRID	=>
								);
	ELSE
		fbWritePersistentData(	START	:=FALSE);
	END_IF

	fbWriteErrorREdge(CLK:=fbWritePersistentData.ERR,Q=>WritePersistentData);
END_METHOD

END_FUNCTION_BLOCK

// ---- 01_Submodules/IO-Link/FB_IoLinkMasterDiagnosis.TcPOU
FUNCTION_BLOCK FB_IoLinkMasterDiagnosis
VAR
	//実I/Oにリンク
	byStatus			AT %I*	:ARRAY[1..8] OF BYTE;		//State Ch.*にリンク
	_bOccurrenceEvent	AT %I*	:BOOL;						//Device Diagにリンク
	_bPortError			AT %I*	:BOOL;						//Device Stateにリンク
	
	//初期化の際に入力
	bEnabledPort				:ARRAY[1..8] OF BOOL;
END_VAR

(*
BeckhoffのIO-Linkマスターで使用する前提のファンクションブロックです。
初期化の際に使用するIO-LinkポートをTRUEにしてください。

デバイスでイベント発生時にはbOccurrenceEventがTRUEになります。
どれかのデバイスと通信が中断した場合にはbPortErrorがTRUEになります。

どのポートにてエラーが発生しているかは、iPortErrorのBitでわかります。
ポート1はBit1,ポート2はBit2。。。ポート8はBit8

ポートのエラーとステータスの内容はメソッドIoLinkPortDiagnosisでわかります。
*)

PROPERTY bOccurrenceEvent : BOOL
GET
bOccurrenceEvent:=_bOccurrenceEvent;
END_GET
END_PROPERTY

PROPERTY bPortError : BOOL
GET
bPortError:=_bPortError;
END_GET
END_PROPERTY

//FB_Init は常に暗黙的に使用可能で、主に初期化に使用されます。
//戻り値は評価されません。特定の結果を得るために、メソッドを明示的に宣言し、
//そのメソッドに標準の初期化コードをもったコードを追加することができます。戻り値を評価できます。
METHOD FB_Init: BOOL
VAR_INPUT
    bInitRetains	:BOOL; // TRUE: 保持変数は初期化されます (ウォーム リセット、あるいはコールド リセット)
    bInCopyCode		:BOOL;  // TRUE: 後でコードをコピーする (オンライン変更) ために、インスタンスをコピーします。
	
	bEnabledPort	:ARRAY[1..8] OF BOOL;
END_VAR
VAR
	i				:INT;
END_VAR
FOR i:=1 TO 8 DO
	THIS^.bEnabledPort[i]:=bEnabledPort[i];
END_FOR
END_METHOD

METHOD IoLinkPortDiagnosis
VAR_INPUT
	eIoLinkPort				:E_IolPort;
	eIoLinkPortError		:REFERENCE TO E_IolPortError;
	eIoLinkPortState		:REFERENCE TO E_IolPortState;
	sChannelStateText		:REFERENCE TO STRING;
END_VAR
eIoLinkPortError	:=F_IolGetPortError(byStatus[eIoLinkPort]);
eIoLinkPortState	:=F_IolGetPortState(byStatus[eIoLinkPort]);
sChannelStateText	:=F_IolGetChannelStateTxt(nIolChState:=byStatus[eIoLinkPort],nPort:=eIoLinkPort);

(*
Port Error
Name					Value
NoError					:0
WatchdogDetected		:1
InternalError			:2
InvalidDeviceID			:3
InvalidVendorID			:4
InvalidIOLinkVersion	:5
InvalidFrameCapability	:6
InvalidCycletime		:7
InvalidPdInLength		:8
InvalidPdOutLenght		:9
NoDeviceDetected		:10

Port State
Name					Value
Disabled				:0
stDigIn					:1
stDigOut				:2
CommunicationOP			:3
CommunicationComstop	:4
*)
END_METHOD

PROPERTY iPortError : int
GET
VAR
	i		:INT;
END_VAR
IF _bPortError=TRUE THEN
	FOR i := 1 TO 8 DO
		IF bEnabledPort[i]=TRUE AND F_IolGetPortError(byStatus[i])<>E_IolPortError.NoError THEN
			CASE  i OF
				1:iPortError.1:=TRUE;
				2:iPortError.2:=TRUE;
				3:iPortError.3:=TRUE;
				4:iPortError.4:=TRUE;
				5:iPortError.5:=TRUE;
				6:iPortError.6:=TRUE;
				7:iPortError.7:=TRUE;
				8:iPortError.8:=TRUE;
			END_CASE
		END_IF	
	END_FOR
END_IF
END_GET
END_PROPERTY

END_FUNCTION_BLOCK

// ---- 01_Submodules/IO-Link/787/FB_787.TcPOU
FUNCTION_BLOCK FB_787 EXTENDS FB_IolStdVarSlave
	VAR CONSTANT
		//チャンネル数
		iNumberChannel						:INT	:=4;
	END_VAR
	VAR_OUTPUT
		bError								:BOOL;
		bWarning							:BOOL;
		bInfo								:BOOL;
	END_VAR
	VAR	
//---プロセスデータとリンク--
		//インプットデータ
		bOff						AT %I*	:BIT;
		bTrippedCollective			AT %I*	:BIT;
		bOver90						AT %I*	:BIT;
		bOver100					AT %I*	:BIT;
		bHardwareFuse				AT %I*	:BIT;
		bLocalOff					AT %I*	:BIT;
		bInputVoltageAlarm			AT %I*	:BIT;
		byControlByteDump			AT %I*	:BYTE;
		byPdByte3					AT %I*	:BYTE;
		byPdByte4					AT %I*	:BYTE;
		byPdByte5					AT %I*	:BYTE;
		//アプトプットデータ
		byChOnOffReset				AT %Q*	:BYTE:=0;
		byControlByte				AT %Q*	:BYTE;
		byValidByte					AT %Q*	:BYTE:=7;

//---サーキットプロテクターの状態確認---
		//負荷状態
		bWarningOverloadOver90Percent		:ARRAY[1..iNumberChannel] OF BOOL;
		bWarningOverloadOver100Percent		:ARRAY[1..iNumberChannel] OF BOOL;
		//トリップ状態
		bTripped							:ARRAY[1..iNumberChannel] OF BOOL;
		bTrippedThermalRelease				:ARRAY[1..iNumberChannel] OF BOOL;
		bTrippedHardwareError				:ARRAY[1..iNumberChannel] OF BOOL;
		//スイッチ状態
		bSwitchedOn							:ARRAY[1..iNumberChannel] OF BOOL;
		bSwitchedOffLocal					:ARRAY[1..iNumberChannel] OF BOOL;
		bSwitchedOffRemote					:ARRAY[1..iNumberChannel] OF BOOL;
		//ブレーカー設定電流
		lrBreakerCurrentSetting				:ARRAY[1..iNumberChannel] OF LREAL;
		//ブレーカーローターリースイッチ設定
		bBreakerRemoteControlSetting		:ARRAY[1..iNumberChannel] OF BOOL;
		//ブレーカーへの入力電圧
		_lrInputVoltage						:LREAL;
		//電流値
		lrActualCurrent						:ARRAY[1..iNumberChannel] OF LREAL;

//---変数---
		//For loop用
		iForIndex							:INT;
		
		//GetAllState用
		iGetStateStep						:INT;
		fbGetStateTimeOut					:TON	:=(PT:=T#2S);
		_bImmediatelyGetInputVoltage		:BOOL;
		bVoltageMsgSent						:BOOL;
		
		//OutputAllError用
		fbInputVoltageAlarmREdge			:R_TRIG;
		fbMessage							:ARRAY[0..iNumberChannel] OF FB_TcMessage;
		
		eNow787Status						:E_787Status;
		ePrev787State						:ARRAY[1..iNumberChannel] OF E_787Status;
	END_VAR

(*
wagoの787-1664/0000-0080で使用するFBです。

初期化の際にIO-LinkマスターのAoE Net IDと接続先ポートナンバーとデバイス名を設定して下さい。
この三項目を設定しないとFB_IolStdVarSlaveのメソッドが使えません。

トリップ、ハードウェアエラー、入力電圧異常(アレイの要素数0)が発生した場合は、bErrorがTRUEになります。
負荷が90%以上、100%以上のチャンネルがある場合は、bWarningがTRUEになります。
リモートOFF、ローカルOFFのチャンネルがある場合は、bInfoがTRUEになります。
各チャンネルがアレイの要素数になります。

各チャンネルのONとOFF、トリップ時のリセットは、ハードのボタンから実施して下さい。
*)

CollectiveMessage();
GetAllState(_bImmediatelyGetInputVoltage);
OutputAllStatus();

METHOD ActualCurrent : LREAL
VAR_INPUT
	iChannel		:INT;
END_VAR
IF iChannel<1 OR iNumberChannel<iChannel THEN
	ActualCurrent:=-1.0;
ELSE
	ActualCurrent:=lrActualCurrent[iChannel];
END_IF
END_METHOD

METHOD BreakerCurrentSetting : LREAL
VAR_INPUT
	iChannel		:INT;
END_VAR
IF iChannel<1 OR iNumberChannel<iChannel THEN
	BreakerCurrentSetting:=-1.0;
ELSE
	BreakerCurrentSetting:=lrBreakerCurrentSetting[iChannel];
END_IF
END_METHOD

METHOD INTERNAL ChannelStatus: E_787Status
VAR_INPUT
	iChannel		:INT;
END_VAR
IF bTrippedHardwareError[iChannel] THEN
	ChannelStatus:=E_787Status.TrippedHardwareError;

ELSIF bTripped[iChannel] THEN
	ChannelStatus:=E_787Status.Tripped;

ELSIF bTrippedThermalRelease[iChannel] THEN
	ChannelStatus:=E_787Status.TrippedThermalRelease;
		
ELSIF bWarningOverloadOver100Percent[iChannel] THEN
	ChannelStatus:=E_787Status.SwitchedOnOverloadOver100Percent;
	
ELSIF bWarningOverloadOver90Percent[iChannel] THEN
	ChannelStatus:=E_787Status.SwitchedOnOverloadOver90Percent;
	
ELSIF bSwitchedOn[iChannel] THEN
	ChannelStatus:=E_787Status.SwitchedOn;
	
ELSIF bSwitchedOffLocal[iChannel] OR bSwitchedOffRemote[iChannel] THEN
	ChannelStatus:=E_787Status.switchedOffLocalOrRemote;
	
ELSE
	ChannelStatus:=E_787Status.InitializationDevice;
	
END_IF
END_METHOD

METHOD INTERNAL CollectiveMessage
bError:=bInputVoltageAlarm OR bHardwareFuse OR bTrippedCollective;

bWarning:=bOver100 OR bOver90;

bInfo:=bOff OR bLocalOff;
END_METHOD

//FB_Init は常に暗黙的に使用可能で、主に初期化に使用されます。
//戻り値は評価されません。特定の結果を得るために、メソッドを明示的に宣言し、
//そのメソッドに標準の初期化コードをもったコードを追加することができます。戻り値を評価できます。
METHOD FB_Init: BOOL
VAR_INPUT
    bInitRetains: BOOL; // TRUE: 保持変数は初期化されます (ウォーム リセット、あるいはコールド リセット)
    bInCopyCode: BOOL;  // TRUE: 後でコードをコピーする (オンライン変更) ために、インスタンスをコピーします。
	
	MasterAoeNetId	:T_AmsNetID;
	port			:E_IolPort;
	Name			:STRING(255);

END_VAR
SUPER^.MasterAoeNetId	:=MasterAoeNetId;
SUPER^.Port				:=port;
SUPER^.Name				:=Name;

//アプトプットデータに念のため書き込み実行
byChOnOffReset	:=0;
byValidByte		:=7;
END_METHOD

METHOD INTERNAL GetAllState
VAR_INPUT
	bImmediatelyGetInputVoltage		:REFERENCE TO BOOL;
END_VAR
//タイムアウト検出
fbGetStateTimeOut();

IF fbGetStateTimeOut.Q THEN
	
	IF __ISVALIDREF(bImmediatelyGetInputVoltage) AND_THEN bImmediatelyGetInputVoltage THEN
		bImmediatelyGetInputVoltage:=FALSE;
	END_IF

	fbGetStateTimeOut.IN:=FALSE;
	iGetStateStep:=0;
END_IF


//電圧異常発生時
IF __ISVALIDREF(bImmediatelyGetInputVoltage) AND_THEN bImmediatelyGetInputVoltage THEN
	fbGetStateTimeOut.IN:=FALSE;
	iGetStateStep:=3;
END_IF


//---ステータスの読み出し---
CASE iGetStateStep OF
	0:	iGetStateStep:=1;//ステイする必要が出来たら追加する
	
	1:	byControlByte:=1;
		fbGetStateTimeOut.IN:=TRUE;
		
		IF byControlByteDump = byControlByte THEN
			bWarningOverloadOver100Percent[1]	:=byPdByte3.0;
			bWarningOverloadOver100Percent[2]	:=byPdByte3.1;
			bWarningOverloadOver100Percent[3]	:=byPdByte3.2;
			bWarningOverloadOver100Percent[4]	:=byPdByte3.3;
			
			bTripped[1]							:=byPdByte4.0;
			bTripped[2]							:=byPdByte4.1;
			bTripped[3]							:=byPdByte4.2;
			bTripped[4]							:=byPdByte4.3;
			
			bSwitchedOffLocal[1]				:=byPdByte5.0;
			bSwitchedOffLocal[2]				:=byPdByte5.1;
			bSwitchedOffLocal[3]				:=byPdByte5.2;
			bSwitchedOffLocal[4]				:=byPdByte5.3;
			
			fbGetStateTimeOut.IN:=FALSE;
			iGetStateStep:=3;
		END_IF

	3:	byControlByte:=3;
		fbGetStateTimeOut.IN:=TRUE;
		
		IF byControlByteDump = byControlByte THEN
			bWarningOverloadOver90Percent[1]	:=byPdByte3.0;
			bWarningOverloadOver90Percent[2]	:=byPdByte3.1;
			bWarningOverloadOver90Percent[3]	:=byPdByte3.2;
			bWarningOverloadOver90Percent[4]	:=byPdByte3.3;
			
			bTrippedHardwareError[1]			:=byPdByte4.0;
			bTrippedHardwareError[2]			:=byPdByte4.1;
			bTrippedHardwareError[3]			:=byPdByte4.2;
			bTrippedHardwareError[4]			:=byPdByte4.3;
			
			_lrInputVoltage						:=(byPdByte5/10.0)+15;
			
			IF __ISVALIDREF(bImmediatelyGetInputVoltage) AND_THEN bImmediatelyGetInputVoltage THEN
				bImmediatelyGetInputVoltage:=FALSE;
			END_IF
			
			fbGetStateTimeOut.IN:=FALSE;
			iGetStateStep:=6;
		END_IF
	
	6:	byControlByte:=6;
		fbGetStateTimeOut.IN:=TRUE;
		
		IF byControlByteDump = byControlByte THEN
			bSwitchedOffRemote[1]				:=byPdByte4.0;
			bSwitchedOffRemote[2]				:=byPdByte4.1;
			bSwitchedOffRemote[3]				:=byPdByte4.2;
			bSwitchedOffRemote[4]				:=byPdByte4.3;
			
			fbGetStateTimeOut.IN:=FALSE;
			iGetStateStep:=13;
		END_IF
	
	13:	byControlByte:=13;
		fbGetStateTimeOut.IN:=TRUE;
		
		IF byControlByteDump = byControlByte THEN
			bSwitchedOn[1]						:=byPdByte3.0;
			bSwitchedOn[2]						:=byPdByte3.1;
			bSwitchedOn[3]						:=byPdByte3.2;
			bSwitchedOn[4]						:=byPdByte3.3;
			
			lrActualCurrent[1]					:=BYTE_TO_LREAL(byPdByte4)/10.0;
			lrActualCurrent[2]					:=BYTE_TO_LREAL(byPdByte5)/10.0;
			
			fbGetStateTimeOut.IN:=FALSE;
			iGetStateStep:=14;
		END_IF
	
	14:	byControlByte:=14;
		fbGetStateTimeOut.IN:=TRUE;
		
		IF byControlByteDump = byControlByte THEN
			lrActualCurrent[3]					:=BYTE_TO_LREAL(byPdByte4)/10.0;
			lrActualCurrent[4]					:=BYTE_TO_LREAL(byPdByte5)/10.0;
			
			fbGetStateTimeOut.IN:=FALSE;
			iGetStateStep:=17;
		END_IF
		
	17:	byControlByte:=17;
		fbGetStateTimeOut.IN:=TRUE;
		
		IF byControlByteDump = byControlByte THEN
			bTrippedThermalRelease[1]			:=byPdByte4.0;
			bTrippedThermalRelease[2]			:=byPdByte4.1;
			bTrippedThermalRelease[3]			:=byPdByte4.2;
			bTrippedThermalRelease[4]			:=byPdByte4.3;
			
			fbGetStateTimeOut.IN:=FALSE;
			iGetStateStep:=18;
		END_IF

	18:	byControlByte:=18;
		fbGetStateTimeOut.IN:=TRUE;
		
		IF byControlByteDump = byControlByte THEN
			lrBreakerCurrentSetting[1]			:=BYTE_TO_LREAL(byPdByte4)/10.0;
			lrBreakerCurrentSetting[2]			:=BYTE_TO_LREAL(byPdByte5)/10.0;
			
			fbGetStateTimeOut.IN:=FALSE;
			iGetStateStep:=19;
		END_IF

	19:	byControlByte:=19;
		fbGetStateTimeOut.IN:=TRUE;
		
		IF byControlByteDump = byControlByte THEN
			lrBreakerCurrentSetting[3]			:=BYTE_TO_LREAL(byPdByte4)/10.0;
			lrBreakerCurrentSetting[4]			:=BYTE_TO_LREAL(byPdByte5)/10.0;
			
			fbGetStateTimeOut.IN:=FALSE;
			iGetStateStep:=22;
		END_IF
		
	22:	byControlByte:=22;
		fbGetStateTimeOut.IN:=TRUE;
		
		IF byControlByteDump = byControlByte THEN
			bBreakerRemoteControlSetting[1]		:=byPdByte4.0;
			bBreakerRemoteControlSetting[2]		:=byPdByte4.1;
			bBreakerRemoteControlSetting[3]		:=byPdByte4.2;
			bBreakerRemoteControlSetting[4]		:=byPdByte4.3;
			
			fbGetStateTimeOut.IN:=FALSE;
			iGetStateStep:=0;
		END_IF

END_CASE
END_METHOD

PROPERTY lrInputVoltage : LREAL
GET
lrInputVoltage:=_lrInputVoltage;
END_GET
END_PROPERTY

METHOD INTERNAL OutputAllStatus
//---ステータスの状態を出力---

//入力電圧異常
	fbInputVoltageAlarmREdge(CLK:=bInputVoltageAlarm);	//異常発生の立ち上がりエッジ検出
	
	//異常発生が立ち上がったらイベントをクリエイト
	IF fbInputVoltageAlarmREdge.Q THEN
		fbMessage[0].CreateEx(TC_EVENTS.TkWagoCp787EventClass.InputVoltageAlarm);
		_bImmediatelyGetInputVoltage:=TRUE;
	END_IF
	
	//
	IF 	bInputVoltageAlarm AND NOT _bImmediatelyGetInputVoltage AND NOT bVoltageMsgSent THEN
		fbMessage[0].ipArguments.Clear().AddLReal(_lrInputVoltage);
		fbMessage[0].Send();
		bVoltageMsgSent:=TRUE;
	ELSIF NOT bInputVoltageAlarm THEN
		fbMessage[0].Release();
		bVoltageMsgSent:=FALSE;
	END_IF

//各チャンネル状態出力
FOR iForIndex := 1 TO iNumberChannel BY 1 DO
	
	//チャンネルのステータスを読み出し
	eNow787Status:=ChannelStatus(iChannel:=iForIndex);
	
	//ステータスが切り替わったらイベントをクリエイト
	IF eNow787Status <> ePrev787State[iForIndex] THEN
		
		CASE eNow787Status OF
		//トリップ状態
		E_787Status.TrippedHardwareError:
			fbMessage[iForIndex].CreateEx(TC_EVENTS.TkWagoCp787EventClass.TrippedHardwareError);
			fbMessage[iForIndex].ipArguments.Clear().AddInt(iForIndex);
			fbMessage[iForIndex].Send();
		
		E_787Status.Tripped,E_787Status.TrippedThermalRelease:
			fbMessage[iForIndex].CreateEx(TC_EVENTS.TkWagoCp787EventClass.Tripped);
			fbMessage[iForIndex].ipArguments.Clear().AddInt(iForIndex);
			fbMessage[iForIndex].Send();
		
		//負荷状態
		E_787Status.SwitchedOnOverloadOver100Percent:
			fbMessage[iForIndex].CreateEx(TC_EVENTS.TkWagoCp787EventClass.OverloadOver100Percent);
			fbMessage[iForIndex].ipArguments.Clear().AddInt(iForIndex);
			fbMessage[iForIndex].Send();
		
		E_787Status.SwitchedOnOverloadOver90Percent:
			fbMessage[iForIndex].CreateEx(TC_EVENTS.TkWagoCp787EventClass.OverloadOver90Percent);
			fbMessage[iForIndex].ipArguments.Clear().AddInt(iForIndex);
			fbMessage[iForIndex].Send();
		
		//スイッチ状態
		E_787Status.switchedOffLocalOrRemote:
			fbMessage[iForIndex].CreateEx(TC_EVENTS.TkWagoCp787EventClass.SwitchedOffLocalOrRemote);
			fbMessage[iForIndex].ipArguments.Clear().AddInt(iForIndex);
			fbMessage[iForIndex].Send();

		//スイッチ状態ON(正常)
		E_787Status.SwitchedOn:
			fbMessage[iForIndex].Release();

		END_CASE
		
	END_IF
	
	//現在のチャンネルステータスを保存
	ePrev787State[iForIndex]:=eNow787Status;
	
END_FOR
END_METHOD

END_FUNCTION_BLOCK

// ---- 01_Submodules/IO-Link/Patlite/FB_IoLinkPatlite.TcPOU
FUNCTION_BLOCK FB_IoLinkPatlite EXTENDS FB_IolStdVarSlave IMPLEMENTS I_Patlite
VAR
	bBuzzerON			AT %Q*	:BOOL;					//ブザー出力
	bRedTier			AT %Q*	:BOOL;					//RedLED出力
	bYellowTier			AT %Q*	:BOOL;					//YellowLED出力
	bGreenTier			AT %Q*	:BOOL;					//GreenLED出力
	bBlueTier			AT %Q*	:BOOL;					//BlueLED出力
	bWhiteTier			AT %Q*	:BOOL;					//WhiteLED出力
	
	bBuzzerFlag					:BOOL;					//ブザー停止記憶
	
	fbStartupBuzzerREdge		:R_TRIG;
	fbStartupBuzzerFEdge		:F_TRIG;
	
	hr							:HRESULT;
	fbhrTon						:ton:=(PT:=T#1S);
	
	usiBuzzerPattern			:USINT;
	usiReadBuzzerPattern		:USINT;

	iStep						:INT;
	ePrevMachineState			:E_MachineState;
	
END_VAR

(*
パトライトのLB6-20ILWCBW用FB

初期化の際にIO-LinkマスターのAoE Net IDと接続先ポートナンバーとデバイス名を設定して下さい。
この三項目を設定しないとFB_IolStdVarSlaveのメソッドが使えません。

*)

PROPERTY bBuzzerStop : BOOL
SET
//---スイッチが押されたらブザー停止---
	IF bBuzzerStop=TRUE THEN
		bBuzzerON:=FALSE;
		bBuzzerFlag:=TRUE;
	END_IF
END_SET
END_PROPERTY

PROPERTY bStartupBuzzer : BOOL
SET
fbStartupBuzzerREdge(CLK:=bStartupBuzzer);
fbStartupBuzzerFEdge(CLK:=bStartupBuzzer);

IF fbStartupBuzzerREdge.Q=TRUE THEN
	iStep:=1;
	usiBuzzerPattern	:=8;		//スイープ音（ヒューン）500ms ON / 500ms OFF
	bBuzzerON:=TRUE;
	bBuzzerFlag:=FALSE;
ELSIF fbStartupBuzzerFEdge.Q=TRUE THEN
	iStep:=1;
	usiBuzzerPattern	:=3;		//高低音（ピポピポ）
	bBuzzerON:=FALSE;
END_IF


//---パラメーターを書き換え---

(*
fbhrTon(IN:= hr=16#203);
IF fbhrTon.Q THEN
	iStep:=iStep +1;
END_IF
*)

CASE iStep OF
	0:
		(*NA*)
	1:
		hr:=SUPER^.Write_UINT8(	nIndex		:=16#07EE,	//Buzzer Pattern
								nSubindex	:=16#00,
								nData		:=usiBuzzerPattern);					

		IF NOT F_IolIsBusy(hr) THEN
				iStep:=2;
		 END_IF
	
	2:
		hr:=SUPER^.Read_UINT8(	nIndex		:=16#07EE,	//Buzzer Pattern
								nSubindex	:=16#00,
								nData		:=usiReadBuzzerPattern);
								
		IF NOT F_IolIsBusy(hr) THEN
			iStep:=3;
		END_IF
	
	3:
		IF usiReadBuzzerPattern<>usiBuzzerPattern THEN
			iStep:=1;
		ELSE
			iStep:=0;
		END_IF

END_CASE
END_SET
END_PROPERTY

PROPERTY eMachineState : E_MachineState
SET
//---マシーンステートごとにパトライトを制御---

	IF ePrevMachineState<>eMachineState THEN
		bBuzzerON:=FALSE;
		bBuzzerFlag:=FALSE;
		ePrevMachineState:=eMachineState;
	END_IF

	CASE eMachineState OF
		
		E_MachineState.Critical:
			IF bBuzzerFlag=FALSE THEN
				bBuzzerON:=TRUE;
			END_IF
		
			bRedTier			:=TRUE;
			bYellowTier			:=FALSE;
			bGreenTier			:=FALSE;
			bBlueTier			:=TRUE;
			bWhiteTier			:=FALSE;
		
		E_MachineState.Error:
			IF bBuzzerFlag=FALSE THEN
				bBuzzerON:=TRUE;
			END_IF
		
			bRedTier			:=TRUE;
			bYellowTier			:=FALSE;
			bGreenTier			:=FALSE;
			bBlueTier			:=FALSE;
			bWhiteTier			:=FALSE;

		E_MachineState.Warning:
			IF bBuzzerFlag=FALSE THEN
				bBuzzerON:=TRUE;
			END_IF
		
			bRedTier			:=FALSE;
			bYellowTier			:=TRUE;
			bGreenTier			:=FALSE;
			bBlueTier			:=FALSE;
			bWhiteTier			:=FALSE;

			
		E_MachineState.Stay:
			bRedTier			:=FALSE;
			bYellowTier			:=FALSE;
			bGreenTier			:=FALSE;
			bBlueTier			:=FALSE;
			bWhiteTier			:=TRUE;
		
		E_MachineState.Stop:
			bRedTier			:=FALSE;
			bYellowTier			:=FALSE;
			bGreenTier			:=TRUE;
			bBlueTier			:=FALSE;
			bWhiteTier			:=TRUE;
	
		E_MachineState.Moving:
			bRedTier			:=FALSE;
			bYellowTier			:=FALSE;
			bGreenTier			:=TRUE;
			bBlueTier			:=FALSE;
			bWhiteTier			:=FALSE;

	END_CASE;
END_SET
END_PROPERTY

//FB_Init は常に暗黙的に使用可能で、主に初期化に使用されます。
//戻り値は評価されません。特定の結果を得るために、メソッドを明示的に宣言し、
//そのメソッドに標準の初期化コードをもったコードを追加することができます。戻り値を評価できます。
METHOD FB_Init: BOOL
VAR_INPUT
    bInitRetains: BOOL; // TRUE: 保持変数は初期化されます (ウォーム リセット、あるいはコールド リセット)
    bInCopyCode: BOOL;  // TRUE: 後でコードをコピーする (オンライン変更) ために、インスタンスをコピーします。
	
	MasterAoeNetId	:T_AmsNetID;
	port			:E_IolPort;
	Name			:STRING(255);

END_VAR
SUPER^.MasterAoeNetId	:=MasterAoeNetId;
SUPER^.Port				:=port;
SUPER^.Name				:=Name;
END_METHOD

END_FUNCTION_BLOCK

// ---- 01_Submodules/PcManagement/1sUPS/FB_1sUPS_BAPI.TcPOU
FUNCTION_BLOCK FB_1sUPS_BAPI IMPLEMENTS i1sUPS
VAR
	fb1sUps		:FB_S_UPS_BAPI;
END_VAR

PROPERTY bPowerFailDetect : BOOL
GET
bPowerFailDetect:=fb1sUps.bPowerFailDetect;
END_GET
END_PROPERTY

PROPERTY eUpsState : E_S_UPS_State
GET
eUpsState := fb1sUps.eState;
END_GET
END_PROPERTY

METHOD UPSCall
VAR_INPUT
	(*PC AMS Net ID*)
	PcAmsNetId	: AMSNETID;
END_VAR
fb1sUps(sNetID				:=F_CreateAmsNetId(PcAmsNetId),
		iPLCPort			:=_AppInfo.AdsPort,
		tTimeout			:=DEFAULT_ADS_TIMEOUT,
		eUpsMode			:=E_S_UPS_Mode.eSUPS_WrPersistData_Shutdown,
		ePersistentMode		:=E_PersistentMode.SPDM_2PASS,
		tRecoverTime		:=T#10S,
		bPowerFailDetect	=>,
		eState				=>,
		nCapacity			=>,
		bBusy				=>,
		bError				=>,
		nErrID				=>
		);
END_METHOD

END_FUNCTION_BLOCK

// ---- 01_Submodules/PcManagement/FB_PcPowerManagement.TcPOU
FUNCTION_BLOCK FB_PcPowerManagement
VAR
	fbWritePersistentData		:FB_WritePersistentData;	//パーシステントデータ書き込み
	
	fbPlcStop					:PLC_Stop;					//PLCストップ
	
	fbNtShutdown				:NT_Shutdown;				//PCシャットダウン
	fbNtReboot					:NT_Reboot;					//PCリブート
	
	fb1sUPS						:i1sUPS;					//1sUPS管理FB
	
	PcAmsNetId					:AMSNETID;					//PC AMS Net ID
	
	fbRebootTon					:TON;
	fbShutdownTon				:TON;
	
	iRebootStep					:INT;
	iShutdownStep				:INT;
END_VAR
VAR PERSISTENT
	bPowerFailDetected			:BOOL;						//停電検知記憶
END_VAR

//FB_Init は常に暗黙的に使用可能で、主に初期化に使用されます。
//戻り値は評価されません。特定の結果を得るために、メソッドを明示的に宣言し、
//そのメソッドに標準の初期化コードをもったコードを追加することができます。戻り値を評価できます。
METHOD FB_Init: BOOL
VAR_INPUT
    bInitRetains: BOOL; // TRUE: 保持変数は初期化されます (ウォーム リセット、あるいはコールド リセット)
    bInCopyCode: BOOL;  // TRUE: 後でコードをコピーする (オンライン変更) ために、インスタンスをコピーします。

	PcAmsNetId			:AMSNETID;		//PC AMS Net ID
	fb1sUPS				:i1sUPS;
END_VAR
THIS^.PcAmsNetId		:=PcAmsNetId;
THIS^.fb1sUPS			:=fb1sUPS;
END_METHOD

METHOD Reboot
VAR_INPUT
	bReboot	:bool;
END_VAR
CASE iRebootStep OF
	0:
		fbRebootTon(IN:=bReboot,PT:=T#2S,Q=>,ET=>);
			
		IF fbRebootTon.Q=TRUE THEN
			fbWritePersistentData.START:=TRUE;
			iRebootStep:=1;			
		END_IF

	1:
		fbWritePersistentData(	NETID	:=F_CreateAmsNetId(PcAmsNetId),
								PORT	:=_AppInfo.AdsPort,
								START	:=,
								TMOUT	:=DEFAULT_ADS_TIMEOUT,
								MODE	:=E_PersistentMode.SPDM_2PASS,
								BUSY	=>,
								ERR		=>,
								ERRID	=>
								);
	
		IF fbWritePersistentData.BUSY=FALSE THEN
			fbWritePersistentData.START:=FALSE;
			iRebootStep:=2;
		END_IF
	
	2:
		fbPlcStop.STOP:=TRUE;
		fbNtReboot.START:=TRUE;
		iRebootStep:=3;
	
	3:
		fbPlcStop(	NETID	:=F_CreateAmsNetId(PcAmsNetId),
					PORT	:=_AppInfo.AdsPort,
					Stop	:=,
					TMOUT	:=DEFAULT_ADS_TIMEOUT,
					BUSY	=>,
					ERR		=>,
					ERRID	=>
					);

		fbNtReboot(	NETID	:=F_CreateAmsNetId(PcAmsNetId),
					DELAY	:=1,
					START	:=,
					TMOUT	:=DEFAULT_ADS_TIMEOUT,
					BUSY	=>,
					ERR		=>,
					ERRID	=>
					);

END_CASE
END_METHOD

METHOD Shutdown
VAR_INPUT
	bShutdown	:BOOL;
END_VAR
CASE iShutdownStep OF
	0:
		fbShutdownTon(IN:=bShutdown,PT:=T#2S,Q=>,ET=>);
	
		IF fbShutdownTon.Q=TRUE THEN
			fbWritePersistentData.START:=TRUE;
			iShutdownStep:=1;			
		END_IF

	1:
		fbWritePersistentData(	NETID	:=F_CreateAmsNetId(PcAmsNetId),
								PORT	:=_AppInfo.AdsPort,
								START	:=,
								TMOUT	:=DEFAULT_ADS_TIMEOUT,
								MODE	:=E_PersistentMode.SPDM_2PASS,
								BUSY	=>,
								ERR		=>,
								ERRID	=>
								);
	
		IF fbWritePersistentData.BUSY=FALSE THEN
			fbWritePersistentData.START:=FALSE;
			iShutdownStep:=2;
		END_IF
	
	2:
		fbPlcStop.STOP:=TRUE;
		fbNtShutdown.START:=TRUE;
		iShutdownStep:=3;
	
	3:
		fbPlcStop(	NETID	:=F_CreateAmsNetId(PcAmsNetId),
					PORT	:=_AppInfo.AdsPort,
					Stop	:=,
					TMOUT	:=DEFAULT_ADS_TIMEOUT,
					BUSY	=>,
					ERR		=>,
					ERRID	=>
					);

		fbNtShutdown(	NETID	:=F_CreateAmsNetId(PcAmsNetId),
						DELAY	:=1,
						START	:=,
						TMOUT	:=DEFAULT_ADS_TIMEOUT,
						BUSY	=>,
						ERR		=>,
						ERRID	=>
						);
	
END_CASE
END_METHOD

METHOD UPSControl
VAR_INPUT
	bPowerFailDetectReset		:BOOL;
END_VAR
fb1sUPS.UPSCall(PcAmsNetId:=PcAmsNetId);

IF fb1sUPS.bPowerFailDetect=TRUE THEN
	bPowerFailDetected		:=fb1sUPS.bPowerFailDetect;
ELSIF bPowerFailDetectReset=TRUE THEN
	bPowerFailDetected		:=FALSE;
END_IF
END_METHOD

END_FUNCTION_BLOCK

// ---- 01_Submodules/FB_FanControl.TcPOU
FUNCTION_BLOCK FB_FanControl
VAR
//-----PWM-----
	uiPwmPeriod					AT %Q*	:UINT :=40;				//PWMの周期,μｓ単位で、FANは25Hz入力なので、40μs設定
	uiPwmOutput					AT %Q*	:UINT :=65535;			//PWMのパルス幅、％単位の入力。初期値はMAX値(100%)を入力
	_rMaxTemp							:REAL;					//PWMのパルス幅を100%にする温度
	_rMinTemp							:REAL;					//PWMのパルス幅を0%にする温度
	_bManualFanSpeed					:BOOL;					//FANマニュアルスピード有効
	_uiManualFanSpeed					:UINT;					//FANマニュアルスピード設定

//-----吸気ファン-----
	bInFanOn					AT %Q*	:BOOL :=TRUE;			//吸気ファン運転、基本回っているように初期値はTRUE
	_iInAirTemp					AT %I*	:INT;					//吸気ファン側の測温抵抗体温度
	usiInFanInputEvent			AT %I*	:USINT;					//入力が500μs中に何回あったか
	udiInFanInputEventTime		AT %I*	:ARRAY[1..10] OF UDINT;	//入力があった時間
	udiInFanPrevEventTime				:UDINT;					//入力があった前回の時間
	udiInFanDeltaTime					:UDINT;					//入力時間の差
	iInFanInputEventCountUp				:INT;					//入力回数をカウント
	_rInFanSpeed						:REAL;					//吸気ファンの回転スピード[rpm]

//-----排気ファン-----
	bOutFanOn					AT %Q*	:BOOL :=TRUE;			//排気ファン運転、基本回っているように初期値はTRUE	
	_iOutAirTemp				AT %I*	:INT;					//排気ファン側の測温抵抗体温度	
	usiOutFanInputEvent			AT %I*	:USINT;					//入力が500μs中に何回あったか
	udiOutFanInputEventTime		AT %I*	:ARRAY[1..10] OF UDINT;	//入力があった時間
	udiOutFanPrevEventTime				:UDINT;					//入力があった前回の時間
	udiOutFanDeltaTime					:UDINT;					//入力時間の差
	iOutFanInputEventCountUp			:INT;					//入力回数をカウント
	_rOutFanSpeed						:REAL;					//排気ファンの回転スピード[rpm]	
	
END_VAR

(*
FANの仕様
メーカー：オリエンタルモーター
型番：MDV925-24S
電圧：24V
電流：0.04A-0.20A(PWMデューティ0%-100%)
回転速度:1500rpm-5000rpm(PWMデューティ0%-100%)

PWM仕様
PWMデューティ比 (％) ＝ TH/T ×100
PWM 周波数25 (kHz) ＝ 1/T


パルスセンサ
1回転あたり2周期の矩形波の信号を出力するセンサです。回転速度の検出ができます。

パルス入力の仕様
ns単位の32bitでタイムスタンプは与えられる
なので、60s中にパルス数で回転数になるので、60.000,000,000nsを,1回転当たり2周期の信号がFANから出力されるので、５回分のタイムスタンプ差のデルタタイムで割り算する


T1℃の時にパルス幅を0%、T2℃の時にパルス幅100%になるように数式作成
y軸をパルス幅に設定、x軸を温度に設定
y=(dパルス幅/d温度)*x+b
y=(100/(T2-T1))*x+b
0=(100/(T2-T1))*T1+b
b=-100*T1/(T2-T1)

y=100*(x-T1)/(T2-T1)
*)

METHOD AirFanOn
VAR_INPUT
END_VAR
//-----ファンの回転数を計算-----
	//吸気ファン
	_rInFanSpeed:=FC_FanSpeedCalc(	usiFanInputEvent		:=usiInFanInputEvent,
									udiFanInputEventTime	:=udiInFanInputEventTime,
									udiFanPrevEventTime		:=udiInFanPrevEventTime,
									udiFanDeltaTime			:=udiInFanDeltaTime,
									iFanInputEventCountUp	:=iInFanInputEventCountUp);
	//排気ファン
	_rOutFanSpeed:=FC_FanSpeedCalc(	usiFanInputEvent		:=usiOutFanInputEvent,
									udiFanInputEventTime	:=udiOutFanInputEventTime,
									udiFanPrevEventTime		:=udiOutFanPrevEventTime,
									udiFanDeltaTime			:=udiOutFanDeltaTime,
									iFanInputEventCountUp	:=iOutFanInputEventCountUp);

//-----測温抵抗体の温度からPWMの出力幅を決定,マニュアルスピードの場合はマニュアルスピードに変更-----
	IF _bManualFanSpeed=TRUE THEN
		uiPwmOutput:=_uiManualFanSpeed;
	ELSIF _rMaxTemp-_rMinTemp<>0 THEN
		uiPwmOutput:=LREAL_TO_UINT(65535*(_iOutAirTemp/10-_rMinTemp)/(_rMaxTemp-_rMinTemp));
	END_IF
END_METHOD

PROPERTY bManualFanSpeed : BOOL
SET
_bManualFanSpeed:=bManualFanSpeed;
END_SET
END_PROPERTY

METHOD PRIVATE FC_FanSpeedCalc : REAL
VAR_INPUT
	usiFanInputEvent				:USINT;							//入力が500μs中に何回あったか
	udiFanInputEventTime			:ARRAY[1..10] OF UDINT;			//入力があった時間
	udiFanPrevEventTime				:REFERENCE TO UDINT;			//入力があった前回の時間
	udiFanDeltaTime					:REFERENCE TO UDINT;			//入力時間の差	
	iFanInputEventCountUp			:REFERENCE TO INT;				//入力回数をカウント
END_VAR
//-----ファンの回転数を計算-----
	CASE usiFanInputEvent OF
		0:
			(*NA*)
		
		1..4:
			IF iFanInputEventCountUp+usiFanInputEvent<=4 THEN
				iFanInputEventCountUp:=iFanInputEventCountUp+usiFanInputEvent;
				
			ELSE
				IF udiFanInputEventTime[5-iFanInputEventCountUp]>udiFanPrevEventTime THEN
					udiFanDeltaTime:=udiFanInputEventTime[5-iFanInputEventCountUp]-udiFanPrevEventTime;
				END_IF
				udiFanPrevEventTime:=udiFanInputEventTime[usiFanInputEvent];
				
				iFanInputEventCountUp:=1;	
				
			END_IF

			
		5..10:
			udiFanDeltaTime:=udiFanInputEventTime[5]-udiFanInputEventTime[1];

			udiFanPrevEventTime:=udiFanInputEventTime[usiFanInputEvent];
			
			iFanInputEventCountUp:=1;
		
	END_CASE
	
	IF udiFanDeltaTime<>0 THEN
		FC_FanSpeedCalc:=60000000000.0/UDINT_TO_REAL(udiFanDeltaTime);
	END_IF
END_METHOD

PROPERTY iInAirTemp : INT
GET
iInAirTemp:=_iInAirTemp;
END_GET
END_PROPERTY

PROPERTY iOutAirTemp : INT
GET
iOutAirTemp:=_iOutAirTemp;
END_GET
END_PROPERTY

PROPERTY rInFanSpeed : REAL
GET
rInFanSpeed:=_rInFanSpeed;
END_GET
END_PROPERTY

PROPERTY rMaxTemp : REAL
SET
_rMaxTemp:=rMaxTemp;
END_SET
END_PROPERTY

PROPERTY rMinTemp : REAL
SET
_rMinTemp:=rMinTemp;
END_SET
END_PROPERTY

PROPERTY rOutFanSpeed : REAL
GET
rOutFanSpeed:=_rOutFanSpeed;
END_GET
END_PROPERTY

PROPERTY uiManualFanSpeed : UINT
SET
_uiManualFanSpeed:=uiManualFanSpeed;
END_SET
END_PROPERTY

END_FUNCTION_BLOCK

// ---- 01_Submodules/Axis/FB_AxisAbsolute.TcPOU
FUNCTION_BLOCK FB_AxisAbsolute
VAR	
	// =============== Done signals ============================
	_bResetDone			:BOOL;					// Status of function block MC_Reset
	_bHaltDone			:BOOL;					// Status of function block MC_Halt
	_bStopDone			:BOOL;					// Status of function block MC_Stop
	_bMoveDone			:BOOL;					// Status of function block MC_MoveAbsolute

	// =============== State variables ========================
	_bStatusEnable		:BOOL;					// Enable feedback
	_bStateError		:BOOL;					// Error signal
	_bMoveCommandAborted:BOOL;					// Status of function block MC_MoveAbsolute	
	_nStateErrorID		:UDINT;					// Error ID
	_bStateMoving		:BOOL;					// Status of moving
	_fStateActPos		:LREAL;					// Actual Position
	
	// =============== Position Velocity, override ============
	_fTargetPosition	:LREAL;					// Target Position 
	_fTargetVelocity	:LREAL;					// Target Velocity
	fOverride 			:LREAL := 100.0;		// Override 100%
	
	// =============== Axis Limit =============================
	_fMaxPosition		:LREAL;					//	MAX Target Position 
	_fMinPosition		:LREAL;					//	MIN Target Position 
	_fMaxVelocity		:LREAL;					//	MAX Target Velocity
	_fMinVelocity		:LREAL;					//	MIN Target Velocity
	
	// =============== Trigger function blocks ================
	fbTriggerReset		:R_TRIG;				// Trigger to recognize rising edge of reset input
	fbTriggerHalt		:R_TRIG;				// Trigger to recognize rising edge of halt input
	fbTriggerStop		:R_TRIG;				// Trigger to recognize rising edge of stop input
	fbTriggerMove		:R_TRIG;
	
	// =============== Axis reference =========================
	AxisRef				:AXIS_REF;				// Axis reference (process data plc/nc)
	
	// =============== Motion function blocks =================
	fbMcPower 			:MC_Power;				// FB for enable and override
	fbMcReset 			:MC_Reset;				// FB to reset axis
	fbMcStop 			:MC_Stop;				// FB to stop axis
	fbMcHalt			:MC_Halt;				// FB to halt axis
	fbMcMove			:MC_MoveAbsolute;		// FB to move axis (Absolute movement)
END_VAR

// =========================================================
;
// =========================================================

PROPERTY bStateEnable : BOOL
GET
bStateEnable := _bStatusEnable;
END_GET
END_PROPERTY

PROPERTY bStateError : BOOL
GET
bStateError:=_bStateError;
END_GET
END_PROPERTY

PROPERTY bStateHaltDone : BOOL
GET
bStateHaltDone := _bHaltDone;
END_GET
END_PROPERTY

PROPERTY bStateMoveCommandAborted : BOOL
GET
bStateMoveCommandAborted:=_bMoveCommandAborted;
END_GET
END_PROPERTY

PROPERTY bStateMoveDone : BOOL
GET
bStateMoveDone:=_bMoveDone;
END_GET
END_PROPERTY

PROPERTY bStateMoving : BOOL
GET
bStateMoving:=_bStateMoving;
END_GET
END_PROPERTY

PROPERTY bStateResetDone : BOOL
GET
bStateResetDone := _bResetDone;
END_GET
END_PROPERTY

PROPERTY bStateStopDone : BOOL
GET
bStateStopDone:=_bStopDone;
END_GET
END_PROPERTY

METHOD Enable
VAR_INPUT
	bEnable		: BOOL;
END_VAR
// =========================================================

fbMCPower(	Enable 			:= bEnable, 
			Enable_Positive	:= bEnable, 
			Enable_Negative	:= bEnable, 
			Override		:= fOverride,
			Axis			:= AxisRef,
			Status			=> _bStatusEnable);
			
IF fbMcPower.Error THEN
	_bStateError		:= TRUE;
	_nStateErrorID 		:= fbMcPower.ErrorID;
END_IF

AxisRef.ReadStatus();

_bStateMoving	:= AxisRef.Status.Moving;

_fStateActPos	:= AxisRef.NcToPlc.ActPos;

// =========================================================
END_METHOD

//FB_Init は常に暗黙的に使用可能で、主に初期化に使用されます。
//戻り値は評価されません。特定の結果を得るために、メソッドを明示的に宣言し、
//そのメソッドに標準の初期化コードをもったコードを追加することができます。戻り値を評価できます。
METHOD FB_Init: BOOL
VAR_INPUT
    bInitRetains: BOOL; // TRUE: 保持変数は初期化されます (ウォーム リセット、あるいはコールド リセット)
    bInCopyCode: BOOL;  // TRUE: 後でコードをコピーする (オンライン変更) ために、インスタンスをコピーします。
	

	fMaxPosition	:LREAL;
	fMinPosition	:LREAL;
	fMaxVelocity	:LREAL;
	fMinVelocity	:LREAL;
END_VAR
	_fMaxPosition:=fMaxPosition;
	_fMinPosition:=fMinPosition;
	_fMaxVelocity:=fMaxVelocity;
	_fMinVelocity:=fMinVelocity;
END_METHOD

PROPERTY fStateActPos : LREAL
GET
fStateActPos:=_fStateActPos;
END_GET
END_PROPERTY

PROPERTY fTargetPosition : LREAL
GET
fTargetPosition:=_fTargetPosition;
END_GET
SET
_fTargetPosition:=LIMIT(_fMinPosition,fTargetPosition,_fMaxPosition);
END_SET
END_PROPERTY

PROPERTY fTargetVelocity : LREAL
GET
fTargetVelocity := _fTargetVelocity;
END_GET
SET
_fTargetVelocity :=LIMIT(_fMinVelocity ,fTargetVelocity,_fMaxVelocity);
END_SET
END_PROPERTY

METHOD Halt
VAR_INPUT
	bDriveHalt		: BOOL;					// Request stop
END_VAR
// =========================================================

IF bDriveHalt THEN
	// Move Execute FALSE
	fbMCMove(	Execute	:= FALSE,
				Axis 	:= AxisRef);
ELSE
	// Reset done signal
	_bHaltDone := FALSE;
END_IF

// Trigger
fbTriggerHalt(CLK := bDriveHalt);

IF fbTriggerHalt.Q THEN
	fbMcHalt(	Execute	:= TRUE,
				Axis 	:= AxisRef);
ELSE
	fbMcHalt(Axis := AxisRef);
END_IF

// Done / Error / Command aborted
IF fbMcHalt.Done OR fbMcHalt.Error OR fbMcHalt.CommandAborted THEN
	_bStateError		:= fbMcHalt.Error;
	_nStateErrorID		:= fbMcHalt.ErrorID;
	_bHaltDone 			:= fbMcHalt.Done;
	
	fbMCMove(	Execute	:= FALSE,
				Axis 	:= AxisRef);
				
	fbMcHalt(	Execute	:= FALSE,
				Axis 	:= AxisRef);
END_IF

// =========================================================
END_METHOD

METHOD MoveAbsolute
VAR_INPUT
	bMove		:REFERENCE TO BOOL; 
END_VAR
// =========================================================

IF bMove=TRUE AND(fbMCMove.Error=FALSE OR fbMcHalt.Execute=FALSE OR fbMcStop.Execute=FALSE) THEN
	fbMCMove(	Execute 		:=TRUE,
				Position		:=_fTargetPosition,
				Velocity 		:= _fTargetVelocity,
				Axis 			:= AxisRef,
				Done			=>_bMoveDone,
				CommandAborted	=>_bMoveCommandAborted);	
ELSE
	fbMCMove(	Axis 			:= AxisRef);	
END_IF

// Error / Command aborted
IF fbMCMove.Done OR fbMCMove.Error OR fbMCMove.CommandAborted THEN
	IF fbMcMove.Error THEN
		_bStateError		:= TRUE;
		_nStateErrorID		:= fbMCMove.ErrorID;
	END_IF
	
	bMove:=FALSE;
	
	fbMCMove(	Execute 	:=FALSE,
				Axis 		:= AxisRef);
END_IF

IF fbMcStop.Execute=TRUE OR fbMcHalt.Execute=TRUE THEN
	bMove:=FALSE;
END_IF
END_METHOD

PROPERTY nStateErrorID : UDINT
GET
nStateErrorID:=_nStateErrorID;
END_GET
END_PROPERTY

METHOD Reset
VAR_INPUT
	bDriveReset		: BOOL;					// Request reset
END_VAR
// =========================================================

IF NOT bDriveReset THEN
	_bResetDone 	:= FALSE;
END_IF

// Trigger
fbTriggerReset(CLK := bDriveReset);

IF fbTriggerReset.Q THEN
	_bResetDone		:= FALSE;
	
	fbMcReset(Execute := TRUE, Axis := AxisRef);
ELSE
	fbMcReset(Axis := AxisRef);
END_IF

// Done / Error
IF fbMcReset.Done OR fbMcReset.Error THEN
	_bStateError		:= fbMcReset.Error;
	_nStateErrorID		:= fbMcReset.ErrorID;
	_bResetDone 		:= fbMcReset.Done;

	fbMcReset(	Execute	:= FALSE,
				Axis 	:= AxisRef);
END_IF

// =========================================================
END_METHOD

METHOD Stop
VAR_INPUT
	bDriveStop		: BOOL;					// Request stop
END_VAR
// =========================================================

IF bDriveStop THEN
	// Move Execute FALSE
	fbMCMove(	Execute	:= FALSE,
				Axis 	:= AxisRef);
ELSE
	// Reset done signal
	_bStopDone := FALSE;
END_IF

// Trigger
fbTriggerStop(CLK := bDriveStop);

IF fbTriggerStop.Q THEN
	fbMcStop(	Execute	:= TRUE,
				Axis 	:= AxisRef);
ELSE
	fbMcStop(Axis := AxisRef);
END_IF

// Done / Error / Command aborted
IF fbMcStop.Done OR fbMcStop.Error OR fbMcStop.CommandAborted THEN
	_bStateError		:= fbMcStop.Error;
	_nStateErrorID 		:= fbMcStop.ErrorID;
	_bStopDone 			:= fbMcStop.Done;
	
	fbMCMove(	Execute	:= FALSE,
				Axis 	:= AxisRef);
				
	fbMcStop(	Execute	:= FALSE,
				Axis 	:= AxisRef);
END_IF

// =========================================================
END_METHOD

END_FUNCTION_BLOCK

// ---- 01_Submodules/Axis/FB_ZAxisAbsolute.TcPOU
FUNCTION_BLOCK FB_ZAxisAbsolute EXTENDS FB_AxisAbsolute
VAR
	_fXAxisActualPosition	:LREAL;					// X Axis Actual Position 
	_fYAxisActualPosition	:LREAL;					// Y Axis Actual Position 
	_fXZPlaneSlope			:LREAL;					//ステージのXZ軸の傾き
	_fYZPlaneSlope			:LREAL;					//ステージのYZ軸の傾き
	
	fbMoveREdge				:R_TRIG;
END_VAR

(*FB_Init は常に暗黙的に使用可能で、主に初期化に使用されます。
戻り値は評価されません。特定の結果を得るために、メソッドを明示的に宣言し、
そのメソッドに標準の初期化コードをもったコードを追加することができます。戻り値を評価できます。*)
METHOD FB_Init : BOOL
VAR_INPUT
	(* TRUE: 保持変数は初期化されます (ウォーム リセット、あるいはコールド リセット)*)
	bInitRetains	: BOOL;
	(* TRUE: 後でコードをコピーする (オンライン変更) ために、インスタンスをコピーします。*)
	bInCopyCode	: BOOL;
	
	fMaxPosition	: LREAL;
	fMinPosition	: LREAL;
	fMaxVelocity	: LREAL;
	fMinVelocity	: LREAL;
	
	fXZPlaneSlope	:LREAL;
	fYZPlaneSlope	:LREAL;
END_VAR
	_fMaxPosition:=fMaxPosition;
	_fMinPosition:=fMinPosition;
	_fMaxVelocity:=fMaxVelocity;
	_fMinVelocity:=fMinVelocity;

	_fXZPlaneSlope:=fXZPlaneSlope;
	_fYZPlaneSlope:=fYZPlaneSlope;
END_METHOD

PROPERTY fXAxisActualPosition : LREAL
SET
_fXAxisActualPosition:=fXAxisActualPosition;
END_SET
END_PROPERTY

PROPERTY fYAxisActualPosition : LREAL
SET
_fYAxisActualPosition:=fYAxisActualPosition;
END_SET
END_PROPERTY

PROPERTY fZAxisAcc : LREAL
GET
fZAxisAcc:=super^.AxisRef.NcToPlc.SetAcc;
END_GET
END_PROPERTY

METHOD MoveAbsolute
VAR_INPUT
		bMove		:REFERENCE TO BOOL; 
END_VAR
VAR
	lrXbuf		:LREAL;
	lrYbuf		:LREAL;
END_VAR
//XZ平面の傾きとX軸の現在ポジションから調整値を計算
lrXbuf:=_fXZPlaneSlope*_fXAxisActualPosition;

//YZ平面の傾きとY軸の現在ポジションから調整値を計算
lrYbuf:=_fYZPlaneSlope*_fYAxisActualPosition;


fbMoveREdge(CLK:=TRUE);

IF fbMoveREdge.Q=TRUE THEN
	SUPER^.fTargetPosition:=SUPER^.fTargetPosition+lrXbuf+lrYbuf;
END_IF

SUPER^.MoveAbsolute(bMove:=bMove);

//もしかしたら、X,Y軸はアクチュアルポジションではなくてターゲットポジションの方がいいかも？？？
END_METHOD

END_FUNCTION_BLOCK

// ---- 01_Submodules/Axis/FB_GripperAbsolute.TcPOU
FUNCTION_BLOCK FB_GripperAbsolute EXTENDS FB_AxisAbsolute
VAR
	_lrAttachmentDiameter			:LREAL;		//アタッチメントの直径
	_lrAttachmentRotationRadius		:LREAL;		//アタッチメントの回転半径
	
	_lrWorkDiameter					:LREAL;		//ワークの直径
	
	lrCalcBufA						:LREAL;		//計算バッファー
	lrCalcBufB						:LREAL;		//計算バッファー

	lrFingerRotationAngle			:LREAL;		//グリップ角度
END_VAR

(*FB_Init は常に暗黙的に使用可能で、主に初期化に使用されます。
戻り値は評価されません。特定の結果を得るために、メソッドを明示的に宣言し、
そのメソッドに標準の初期化コードをもったコードを追加することができます。戻り値を評価できます。*)
METHOD FB_Init : BOOL
VAR_INPUT
	(* TRUE: 保持変数は初期化されます (ウォーム リセット、あるいはコールド リセット)*)
	bInitRetains	: BOOL;
	(* TRUE: 後でコードをコピーする (オンライン変更) ために、インスタンスをコピーします。*)
	bInCopyCode	: BOOL;
	
	fMaxPosition	: LREAL;
	fMinPosition	: LREAL;
	fMaxVelocity	: LREAL;
	fMinVelocity	: LREAL;
	
	lrAttachmentDiameter			:LREAL;		//アタッチメントの直径
	lrAttachmentRotationRadius		:LREAL;		//アタッチメントの回転半径
END_VAR
	_fMaxPosition:=fMaxPosition;
	_fMinPosition:=fMinPosition;
	_fMaxVelocity:=fMaxVelocity;
	_fMinVelocity:=fMinVelocity;
	
	_lrAttachmentDiameter		:=lrAttachmentDiameter;
	_lrAttachmentRotationRadius	:=lrAttachmentRotationRadius;
END_METHOD

PROPERTY lrWorkDiameter : LREAL
SET
_lrWorkDiameter:=lrWorkDiameter;
END_SET
END_PROPERTY

METHOD WorkGrippingAbs
VAR_INPUT
	bMove		:REFERENCE TO BOOL; 
END_VAR
//ワークの直径からワークをグリップする角度を計算
	lrCalcBufA:=EXPT((_lrWorkDiameter+_lrAttachmentDiameter)/2,2)-EXPT(9.05,2)-EXPT(_lrAttachmentRotationRadius,2);
	lrCalcBufB:=2*9.05*_lrAttachmentRotationRadius;

	IF -1<lrCalcBufA/lrCalcBufB AND lrCalcBufA/lrCalcBufB<1 THEN
		lrFingerRotationAngle:=180/PI*ACOS(lrCalcBufA/lrCalcBufB);
	ELSE
		lrFingerRotationAngle:=0;	//角度計算できない場合噛みこまないように0度にする
	END_IF;
	
//駆動命令起動
	SUPER^.fTargetPosition:=lrFingerRotationAngle;
	SUPER^.MoveAbsolute(bMove:=bMove);
END_METHOD

END_FUNCTION_BLOCK

// ---- 01_Submodules/LoadCell/CalcLoadCell/FB_LoadCell_ForCalcValue.TcPOU
FUNCTION_BLOCK FB_LoadCell_ForCalcValue
VAR PERSISTENT
	_lrTareWeight					:LREAL;													//風袋重量[kg]
END_VAR
VAR
	rRMBValueInput			AT %I*	:ARRAY[1..Param_CalcLoadCell.iOverSamples] OF REAL;		//EtherCATターミナルからの入力
	tTimestamp				AT %I*	:T_DCTIME64;											//EtherCATターミナルからのTimestamp
	_rEexcitationVoltage	AT %Q*	:REAL;													//ロードセル印加電圧 [V] 							
	bSampleMode				AT %Q*	:BOOL	:=TRUE;											//EL3356-0010のConversion mode 0=7.2ms 1=0.72ms latency

	_lrCalibrationWeight			:LREAL;													//校正重量[kg]		
	_lrGrossWeight					:LREAL;													//測定重量[kg]
	_lrNetWeight					:LREAL;													//正味重量[kg]
	lrSlope							:LREAL;													//校正後の傾き
	_lrZAxisSetAcc					:LREAL;													//Z軸の設定加速度[mm/s2]
	i								:INT;													//演算用

	_bError							:BOOL;
	_ipResultMessage				:I_TCMessage;

	// --- TF3685：設定構造体 ---
    _stParamsComboFilter			:ST_WG_ComboFilter;
	_stParamsScale					:ST_WG_Scaling;
  	_stParamsWeighing				:ST_WG_Weighing;
	
	// --- TF3685：FBインスタンス ---
	fbComboFilter 					:FB_WG_ComboFilter;
	fbScale 						:FB_WG_Scaling;
	fbWeighing						:FB_WG_Weighing;

	//-----中間の変数-----
	aInput							:ARRAY[1..Param_CalcLoadCell.iOverSamples] OF LREAL;
	aOutFilter						:ARRAY[1..Param_CalcLoadCell.iOverSamples] OF LREAL;
	aOutScaling						:ARRAY[1..Param_CalcLoadCell.iOverSamples] OF LREAL;



// --- 過去のデータを保存しておくための棚（履歴バッファ） ---
    // 0.5ms(2000Hz)周期で301要素持つことで、150ms分までの過去を記録可能
    alrAccHistory    				:ARRAY[0..300] OF LREAL;								//加速度指令値(Set値)の履歴
    anTimeHistory					:ARRAY[0..300] OF T_DCTIME64;							//その時のDC時刻(Timestamp)の履歴
	
    tDelayOffset     				:T_DCTIME64 := 108*1000000;								//ScopeのTime Markerで測った遅延時間
    _lrGripperWeight				:LREAL;													//グリッパー重量
    
    // --- 計算の過程で使う一時的な変数 ---
	tSearchTime      : T_DCTIME64;              // 「今」から108ms遡った「ターゲットとなる過去の時刻」
	lrTargetAcc      : LREAL;                // 検索で見つけ出した「108ms前の加速度」
	lrCompValue      : LREAL;                // 計算された慣性力（引くべき重さの変動分）
	fCorrectedWeight : LREAL;                // 【最終出力】揺れを打ち消した後の真の重量
	
	fFraction        : LREAL;                // 107.6msなど、ステップ間(0.5ms)の隙間を埋めるための比率
	tDiff            : LREAL;                // 記録されているデータ点同士の時間間隔
END_VAR

METHOD BackgroundCalc
//------EtherCATターミナルからの読み出しデータをアレイへ------
	FOR i := 1 TO Param_CalcLoadCell.iOverSamples BY 1 DO
		aInput[i]:=REAL_TO_LREAL(rRMBValueInput[i]);
	END_FOR

//------TF3685のライブラリーで計算------
	IF NOT fbComboFilter.Call(ADR(aInput), SIZEOF(aInput), ADR(aOutFilter), SIZEOF(aOutFilter)) THEN
		SetError(fbComboFilter);
	END_IF
	
	IF NOT fbScale.Call(ADR(aOutFilter), SIZEOF(aOutFilter), ADR(aOutScaling), SIZEOF(aOutScaling)) THEN
		SetError(fbScale);
	END_IF
	
	IF NOT fbWeighing.Call(ADR(aOutScaling), SIZEOF(aOutScaling)) THEN
		SetError(fbWeighing);
	END_IF

//------履歴の更新------
	//最新データを配列の先頭に入れ、古いものを1つずつ押し出す
	FOR i := 300 TO 1 BY -1 DO
		alrAccHistory[i]:=alrAccHistory[i-1];
		anTimeHistory[i]:=anTimeHistory[i-1];
	END_FOR

	// 配列の[0]に最新の値を格納
	alrAccHistory[0]:=_lrZAxisSetAcc/1000;
	anTimeHistory[0]:=F_GetActualDcTime64();

//------108ms前の加速度をピンポイントで特定する------
	// 「今の時間」から「108ms」を引き算して、探すべき時間を決める
	tSearchTime := anTimeHistory[0] - tDelayOffset; 
	lrTargetAcc := 0;

	FOR i := 1 TO 300 DO
		// 配列の中で、ターゲットの時間を「またいでいる」2点（i番目とi-1番目）を探す
		IF anTimeHistory[i] <= tSearchTime AND anTimeHistory[i-1] > tSearchTime THEN
			
			// その2点間の実際の時間差（通常は周期の0.5msになるはず）
			tDiff := TO_LREAL(anTimeHistory[i-1] - anTimeHistory[i]);
			
			IF tDiff > 0 THEN
				// ターゲット時刻が、その2点間のどこに位置するかを0.0〜1.0で算出（線形補間）
				// 例：107.5ms(i) と 108.0ms(i-1) の間にある 107.6ms を探すため
				fFraction := TO_LREAL(tSearchTime - anTimeHistory[i]) / tDiff;
				
				// 2点の加速度データから、比率(fFraction)を使って間の値を計算
				lrTargetAcc := alrAccHistory[i] + fFraction * (alrAccHistory[i-1] - alrAccHistory[i]);
			ELSE
				// 万が一時間差が取れない場合は、古い方の値を採用
				lrTargetAcc := alrAccHistory[i];
			END_IF
			EXIT; // 見つかったのでループを抜ける
		END_IF
	END_FOR

// ============================================================
// 3. 慣性力の計算と引き算（ここが物理の法則）
// ============================================================
// 物理式：F = m * a  (力 = 質量 * 加速度)
// 単位を合わせるため、標準重力加速度 9.80665 で割って「g」に換算
lrCompValue := (_lrGripperWeight * lrTargetAcc / 9.80665);

// TF3685で綺麗にフィルタリングされた後の重量値から、108ms前の慣性力を引く
fCorrectedWeight := fbWeighing.fWeight + lrCompValue;
END_METHOD

PROPERTY bError : BOOL
GET
bError:=_bError;
END_GET
END_PROPERTY

METHOD CalibrationWeightSet
VAR_INPUT
	bCalibrationWeightSet	:BOOL;
END_VAR
VAR
	lrNowGrossWeight		:LREAL;
END_VAR
	IF bCalibrationWeightSet=TRUE THEN
		
		//今のグロスウェイト確認[kg]
		lrNowGrossWeight:=fbWeighing.fWeight / -1000;

		
		//今のグロスウェイトが風袋重量より重いことを確認
		IF _lrTareWeight+0.010 < lrNowGrossWeight THEN
			//切片を計算
			IF lrNowGrossWeight<>0 AND _lrTareWeight<>0 THEN
				lrSlope:=(_lrCalibrationWeight-0)/(lrNowGrossWeight-_lrTareWeight);
			END_IF
		END_IF
		
	END_IF
END_METHOD

//FB_Init は常に暗黙的に使用可能で、主に初期化に使用されます。
//戻り値は評価されません。特定の結果を得るために、メソッドを明示的に宣言し、
//そのメソッドに標準の初期化コードをもったコードを追加することができます。戻り値を評価できます。
METHOD FB_Init: BOOL
VAR_INPUT
    bInitRetains: BOOL; // TRUE: 保持変数は初期化されます (ウォーム リセット、あるいはコールド リセット)
    bInCopyCode: BOOL;  // TRUE: 後でコードをコピーする (オンライン変更) ために、インスタンスをコピーします。
	
  	stParamsComboFilter		:ST_WG_ComboFilter;
	stParamsScale			:ST_WG_Scaling;
  	stParamsWeighing		:ST_WG_Weighing;
	
	rEexcitationVoltage		:REAL;
	
	lrGripperWeight			:LREAL;
END_VAR
IF bInCopyCode = FALSE THEN

	_stParamsComboFilter	:=stParamsComboFilter;
	_stParamsScale			:=stParamsScale;
	_stParamsWeighing		:=stParamsWeighing;
	
	fbComboFilter.Configure(stConfig:=_stParamsComboFilter);
	fbScale.Configure(stConfig:=_stParamsScale);
	fbWeighing.Configure(stConfig:=_stParamsWeighing);

	_rEexcitationVoltage:=rEexcitationVoltage;

	_lrGripperWeight:=lrGripperWeight;
END_IF
END_METHOD

PROPERTY ipResultMessage : I_TcMessage
GET
ipResultMessage:=_ipResultMessage;
END_GET
END_PROPERTY

PROPERTY lrCalibrationWeight : LREAL
SET
_lrCalibrationWeight:=lrCalibrationWeight;
END_SET
END_PROPERTY

PROPERTY lrGrossWeight : LREAL
GET
//グロスウェイト計算[kg]
	_lrGrossWeight:=fbWeighing.fWeight * 1000.0;
	
	lrGrossWeight:=_lrGrossWeight;
END_GET
END_PROPERTY

PROPERTY lrNetWeight : LREAL
GET
	//ネットウェイト計算[kg]
	_lrNetWeight:=_lrGrossWeight-_lrTareWeight;
	
	lrNetWeight:=_lrNetWeight;
END_GET
END_PROPERTY

PROPERTY lrTareWeight : LREAL
GET
lrTareWeight:=_lrTareWeight;
END_GET
END_PROPERTY

PROPERTY lrZAxisSetAcc : LREAL
SET
_lrZAxisSetAcc:=lrZAxisSetAcc;
END_SET
END_PROPERTY

METHOD Reconfigure
VAR_INPUT
	bReconfigureExe			:REFERENCE TO BOOL;	

  	stParamsComboFilter		:ST_WG_ComboFilter;
	stParamsScale			:ST_WG_Scaling;
  	stParamsWeighing		:ST_WG_Weighing;
END_VAR
IF bReconfigureExe= TRUE THEN

	_stParamsComboFilter	:=stParamsComboFilter;
	_stParamsScale			:=stParamsScale;
	_stParamsWeighing		:=stParamsWeighing;
	
	IF fbComboFilter.Configure(stConfig:=_stParamsComboFilter)=FALSE THEN
		SetError(fbComboFilter);
	ELSIF fbScale.Configure(stConfig:=_stParamsScale)=FALSE THEN
		SetError(fbScale);
	ELSIF fbWeighing.Configure(stConfig:=_stParamsWeighing)=FALSE THEN
		SetError(fbWeighing);
	ELSE
		;
	END_IF
	
	bReconfigureExe:=FALSE;
	
END_IF
END_METHOD

METHOD SetError : BOOL
VAR_INPUT
	fb : REFERENCE TO _FB_WG_BasicImplementationAlgorithm;
END_VAR
THIS^._bError := fb.bError;
THIS^._ipResultMessage := fb.ipResultMessage;
END_METHOD

METHOD TareWeightSet
VAR_INPUT
	bTareWeightSet					:BOOL;
	bPersistentDataWriteRequest		:REFERENCE TO BOOL;
END_VAR
	//風袋重量セット[kg]	
	IF bTareWeightSet=TRUE THEN
		_lrTareWeight:=fbWeighing.fWeight / -1000;
		bPersistentDataWriteRequest:=TRUE;
		
	ELSE
		bPersistentDataWriteRequest:=FALSE;
	END_IF
END_METHOD

END_FUNCTION_BLOCK

// ---- 04_Application/Vision/P_Vision.TcPOU
PROGRAM P_Vision
VAR
	bBlobExecution		:BOOL	:=FALSE;

	bTF7820Execution	:BOOL	:=FALSE;
	bTF3820Execution	:BOOL	:=FALSE;
END_VAR

IF bBlobExecution=TRUE AND bTF7820Execution=FALSE AND bTF3820Execution=FALSE THEN
	P_BlobVision();
ELSIF bBlobExecution=FALSE AND bTF7820Execution=TRUE AND bTF3820Execution=FALSE THEN
	P_DNNVision();
ELSIF bBlobExecution=FALSE and bTF7820Execution=FALSE AND bTF3820Execution=TRUE THEN
	P_MLSVision();
END_IF

END_PROGRAM

// ---- 04_Application/Vision/P_BlobVision.TcPOU
PROGRAM P_BlobVision
VAR
	hr					: HRESULT;					// Vision関数の戻り値を表す変数
	hrTemp				: HRESULT;					// 関数戻り値

	fbCamera			: FB_VN_SimpleCameraControl;// Cameraオブジェクト or File Sourceオブジェクト
	eState				: ETcVnCameraState;			// Cameraオブジェクト (or FileSourceオブジェクト) の状態を表す

	// Images
	ipImageIn			: ITcVnImage;				// 入力画像
	ipImageRes			: ITcVnImage;				// 結果画像
	ipImageProc			: ITcVnImage;				// 途中経過画像
	
	// Displayable Images
	ipImageInDisp		: ITcVnDisplayableImage;	// 入力画像の画面表示用変数
	ipImageResDisp		: ITcVnDisplayableImage;	// 結果画像の画面表示用変数
	ipImageProcDisp		: ITcVnDisplayableImage;	// 途中経過画像1の画面表示用変数
	
	// その他ローカル変数
	nNewImageCounter	: UINT;						// 画像取得カウンタ
	bNewImageArrived	: BOOL;						// 画像取得すると TRUE  (※TRUEの後、すぐにFALSEに戻す)
	bSoftWareTrigger	: BOOL;						// ソフトウェアトリガー
	fbR_TRIG			: R_TRIG;					// ボタンスイッチの立ち上がりエッジを検出
	fbTon				: ton;						// LEDライト点灯安定待ち
	stImageInfo			: TcVnImageInfo;			// 画像情報構造体
	iStep				: INT:=0;					// 画像処理のステップ進行用
	iImageCount			: INT:=0;					// 画像の枚数をカウント用
	
	// ブロブ検出用
	stBlobParams		: TcVnParamsBlobDetection;	// Blob params
	ipContourList		: ITcVnContainer;			// Blob Container
	ipContour			: ITcVnContainer;			// Blob個々の輪郭情報
	ipIterator			: ITcVnForwardIterator;		// 個々のBlobが格納されたコンテナから各要素へアクセスする為のイテレータ （≒ポインタ）	

	fArea				: LREAL;					// 面積 [pixel]

	fbFormatString		: FB_FormatString;			// (need library : "Tc2_Utilities")
	sText				: STRING;
	aDrawPos			: ARRAY[0..1] OF UDINT;
	
	// カラー定義
	aColorRed			: TcVnVector4_LREAL := [255, 50, 50, 0];
	aColorGreen			: TcVnVector4_LREAL := [0, 255, 0, 0];
	aColorBlue			: TcVnVector4_LREAL := [0, 0, 255, 0];
	aColorWhite			: TcVnVector4_LREAL := [255, 255, 255, 0];

END_VAR

eState := fbCamera.GetState();

CASE eState OF
TCVN_CS_ERROR:
	hr := fbCamera.Reset();	// エラーの時はリセットを実行

TCVN_CS_TRIGGERING:
	hr := fbCamera.TriggerImage();	// ソフトウェアトリガー

TCVN_CS_INITIAL..TCVN_CS_STARTACQUISITION:
	hr := fbCamera.StartAcquisition();	// 取込開始状態に移行させる

TCVN_CS_ACQUIRING:

	CASE iStep OF
	0:
		fbR_TRIG(CLK := GVL.bAutoCameraTriger, Q => );	// ボタンスイッチを押すとソフトウェアトリガーを発行する
		
		IF fbR_TRIG.Q=TRUE THEN
			GVL.bLedLight:=TRUE;
		END_IF

		fbTon(IN:=GVL.bLedLight,PT:=T#500MS,Q=>,ET=>);	//LEDの照度安定待ち
		
		IF fbTon.Q=TRUE THEN
			bSoftWareTrigger:=TRUE;
			iStep := 1;
		END_IF
		
	1:
		IF bSoftwareTrigger=TRUE THEN
			hr := fbCamera.TriggerImage();
			IF SUCCEEDED(hr)=TRUE THEN
				bSoftwareTrigger := FALSE;
			END_IF
		ELSE
			hr := fbCamera.GetCurrentImage(ipImageIn);	// 最新画像を取得			
			// new image was received.
			IF SUCCEEDED(hr)=TRUE AND ipImageIn <> 0 THEN
				nNewImageCounter := nNewImageCounter + 1;
				iStep := 2;
			END_IF
		END_IF
		
	2:
			GVL.bLedLight:=FALSE;
			iStep:=3;
	
	3:	
		// Bayerフォーマットからカラー画像へ変換
		// ※画像情報をチェックし、ピクセルフォーマットがBayerエンコーディングされている時はカラー画像に変更。
		// ※最初からカラー画像の時はカラー変換しない。
		hr := F_VN_GetImageInfo(ipImageIn, stImageInfo, hr);
		IF SUCCEEDED(hr) AND_THEN stImageInfo.stPixelFormat.ePixelEncoding <> ETcVnPixelEncoding.TCVN_PE_NONE THEN
			hr := F_VN_ConvertColorSpace(ipImageIn, ipImageIn, TCVN_CST_BAYER_RG_TO_RGB, hr);
		END_IF
		iStep:=4;
	
	4:
		hr := F_VN_CopyImage(ipImageIn, ipimageRes, hr);	// copy to ResultImage
		iStep:=5;
	
	5:
		// グレー画像に変換
		hr := F_VN_ConvertColorSpace(ipImageIn, ipImageProc, ETcVnColorSpaceTransform.TCVN_CST_RGB_TO_GRAY, hr);
		iStep:=6;
		
	6:
		// ブロブ検出パラメータをセット
		stBlobParams.bFilterByArea := TRUE;
		stBlobParams.fMinArea := 1200;
		stBlobParams.fMaxArea := 2500;
		
		// 円形度判別
		stBlobParams.bFilterByCircularity := TRUE;
		stBlobParams.fMinCircularity := 0.70;
		
		// 輝度閾値
		stBlobParams.fMinThreshold	:= 180;
		stBlobParams.fMaxThreshold := 255;
		stBlobParams.fThresholdStep := 0;
		
		// Detect Blobs
		hr := F_VN_DetectBlobs(ipImageProc, ipContourList, stBlobParams, hr);
		
		IF SUCCEEDED(hr) AND ipContourList <> 0 THEN
			hr := ipContourList.GetElementNum(GVL.nDetectedNum);	// 検出したブロブ数を取得
		END_IF
		iStep:=7;

	7:
		IF GVL.nDetectedNum > 0 THEN
			// 検出したブロブの輪郭を描画
			hr := F_VN_DrawContours(ipContourList, -1, ipImageRes,  aColorGreen, 3, hr);
			
			// 各ブロブ情報が格納されたコンテナ(ContourList)から、最初の要素へのイテレータを取得
			hr := F_VN_GetForwardIterator(ipContourList, ipIterator, hr);
			
			//画像のカウンターをリセットする
			iImageCOunt:=0;
			
			WHILE SUCCEEDED(hr) AND_THEN ipIterator.CheckIfEnd() <> S_OK DO
				//画像のカウントをインクリメント
				iImageCount:=iImageCount+1;	
				//アレイの数が10までしか用意してないので、ブロブの検出数が多かった場合は、いったん0に巻き戻す
				IF 10<iImageCount THEN
					iImageCount:=0;
				END_IF
			
				// イテレータが指し示しているContourを取り出す。その後イテレータが次のContourを指し示すよう進める
				hr := F_VN_GetContainer(ipIterator, ipContour, hr);
				hr := F_VN_IncrementIterator(ipIterator, hr);
				
				// Containerから欲しい結果を取得
				hr := F_VN_ContourArea(ipContour, fArea, hr);
				hr := F_VN_ContourCenterOfMass(ipContour, GVL.aMassCenter[iImageCount], hr);
				
				// 個々の結果を描画
				aDrawPos[0] := LREAL_TO_UDINT(GVL.aMassCenter[iImageCount][0]);
				aDrawPos[1] := LREAL_TO_UDINT(GVL.aMassCenter[iImageCount][1]);
				
				// 重心位置をマーク
				hrTemp := F_VN_DrawPointExp(aDrawPos[0], aDrawPos[1], 
											ipImageRes, 
											ETcVnDrawShape.TCVN_DS_PLUS, 
											aColorGreen, 5, 1, 
											ETcVnLineType.TCVN_LT_4_CONNECTED, 0);
				
				// 面積値を結果画像に対して出力
				sText := CONCAT('Area : ', DINT_TO_STRING(LREAL_TO_DINT(fArea)));
				hrTemp := F_VN_PutText(	sText, 
										ipImageRes, 
										aDrawPos[0] - 50, aDrawPos[1] + 20, 
										ETcVnFontType.TCVN_FT_HERSHEY_TRIPLEX, 0.5, aColorRed, 0);
				
				// 座標情報を結果画像に対して出力
				fbFormatString(	sFormat := '(X, Y) = (%0.3f, %0.3f)', 
								arg1 := F_LREAL(GVL.aMassCenter[iImageCount][0]), arg2 := F_LREAL(GVL.aMassCenter[iImageCount][1]), sOut => sText);
				hrTemp := F_VN_PutText(	sText, 
										ipImageRes, 
										aDrawPos[0] - 110, aDrawPos[1] + 40, 
										ETcVnFontType.TCVN_FT_HERSHEY_TRIPLEX, 0.5, aColorRed, 0);
			END_WHILE
			
			FW_SafeRelease(ADR(ipContour));		// ループの外で開放するほうが効率的なので、ここで開放する
			FW_SafeRelease(ADR(ipIterator));	
		END_IF
		FW_SafeRelease(ADR(ipContourList));
							
		istep:=8;
	
	8:		
		// 画面表示イメージを作成する
		hr := F_VN_TransformIntoDisplayableImage(ipImageIn, ipImageInDisp, hr);
		hr := F_VN_TransformIntoDisplayableImage(ipImageRes, ipImageResDisp, S_OK);
		hr := F_VN_TransformIntoDisplayableImage(ipImageProc, ipImageProcDisp, S_OK);
		
		istep:=0;
		
		GVL.bGetImageEnd:=TRUE;
	END_CASE
END_CASE

END_PROGRAM

// ---- 04_Application/Vision/P_DNNVision.TcPOU
PROGRAM P_DNNVision
VAR CONSTANT
	//カメラの画素数
	cImageWidth							:REAL	:=816.0;									//カメラ生画像の幅
    cImageHeight						:REAL	:=624.0;									//カメラ生画像の高さ
	
	//DNNモデルロード用
	cFolderPath							:STRING(255)	:='C:\TF7xxx_NeuralNetwork\';		//ONNXファイルのディレクトリ
	cFileName							:STRING(255)	:='model_InDecode.onnx';			//ONNXファイル名

    //画像とモデルの解像度定義
    cModelInputWidth					:UDINT	:=640;										//ONNXモデルが要求する幅
    cModelInputHeight					:UDINT	:=640;										//ONNXモデルが要求する高さ
	
	//ONNXモデルリターン
	cBatchSize							:UDINT	:=1;										//バッチ数
    cNumBox								:UDINT	:=8400;										//ボックス数
    cElementPerBox						:UDINT	:=6;										//要素数	[cx, cy, w, h, obj_score, class_score]
	
	//ワーク幅
	cWorkWidthMin						:DINT	:=35;										//ワーク幅下限
	cWorkWidthMax						:DINT	:=50;										//ワーク幅上限
END_VAR
VAR
	//制御変数
	nIdx								:UDINT;												//ループ用
	iStep								:INT	:=0;										//画像処理のステップ進行用

	//カメラ・ライト制御
	bSoftWareTrigger					:BOOL;												//ソフトウェアトリガー
	fbR_TRIG							:R_TRIG;											//ボタンスイッチの立ち上がりエッジを検出
	fbTon								:ton;												//LEDライト点灯安定待ち

	//Vision必須関数
    hr									:HRESULT;											//Vision関数の戻り値を表す変数
    fbCameraControl						:FB_VN_SimpleCameraControl;							//Cameraオブジェクト or FileSourceオブジェクト
    eCameraState						:ETcVnCameraState;									//Cameraオブジェクト or FileSourceオブジェクト の状態
	
	//ポストプロセッシングで使用する倍率
	fScale								:REAL;												//レターボックスの縮小倍率
    fPadX								:REAL;												//X方向の余白（ピクセル）
    fPadY								:REAL;												//Y方向の余白（ピクセル）
	
    //DNNモデルロード用
	sFilePath							:STRING(255);										//ONNXファイルのファイルパス
	fbReadDnn							:FB_VN_ReadNeuralNetwork;							//ONNXファイル読み込みFB
	ipDnnModel							:ITcVnNeuralNetwork;								//ONNXのインターフェースポインター
	bDnnModelInitialized				:BOOL	:=FALSE;									//読み込み制御__________________________________後々はFB_Initにする
	nReturnCode							:UDINT;												//リターンコード
	
	
	//DNNモデルインフォメーション
	eInterpolationType					:ETcVnInterpolationType	:=TCVN_IT_BILINEAR;
	ePaddingMode						:ETcVnPaddingMode	:=TCVN_PM_LETTERBOX;
	aGray								:TcVnVector4_LREAL	:=[114, 114, 114, 0];			//グレー(レターボックス塗りつぶし色)
	
    //イメージ
    ipImageIn							:ITcVnImage;										//カメラからの生画像（816x624）
    ipTensorImage						:ITcVnImage;										//前処理（リサイズやREAL化）を施すテンソル
    ipDnnOutputImage	  				:ITcVnImage;										//ONNX実行結果
	ipImageOut							:ITcVnImage;										//結果の画像
	
	//表示用イメージ
	ipImageInDisp						:ITcVnDisplayableImage;								//入力画像の画面表示用変数
	ipImageOutDisp						:ITcVnDisplayableImage;								//結果画像の画面表示用変数

    //Row Data
    aDnnRawOutput						:ARRAY[0..cBatchSize-1, 0..cNumBox-1, 0..cElementPerBox-1] OF REAL;
																							//ONNX生出力受け取り用配列
	//RowData書き込みコンテナ
	ipBoundingBoxes     				:ITcVnContainer;									//座標用コンテナ	(ContainerType_Vector_TcVnRectangle_DINT)
    ipScores            				:ITcVnContainer;									//スコア用コンテナ	(ContainerType_Vector_REAL)

    //コンテナアクセス用
    ipIterator							:ITcVnForwardIterator;								//イテレータ
    ipAccessTcVnRectangleDINT			:ITcVnAccess_TcVnRectangle_DINT;					//アクセスインターフェース(TcVnRectangle_DINT)
	ipAccessREAL						:ITcVnAccess_REAL;									//アクセスインターフェース(REAL)
	stRectangle							:TcVnRectangle_DINT;								//アクセスインターフェースに書き込む中間バッファ
	nIteratorIdx						:DINT;												//イテレータと一緒にカウント
	
	//NMS処理用
	ipDestIndices						:ITcVnContainer;									//NMSで残ったインデックス番号用コンテナ	(ContainerType_Vector_DINT)
	nElementsFound						:ULINT;												//NMSで生き残った確定ワーク数
	
	//結果の出力用
	nTargetIndex						:DINT;												//NMSで生き残った元のインデックス番号
	stFinalRect							:TcVnRectangle_DINT;								//最終確定したワークの座標
	fFinalScore							:REAL;												//最終確定したワークのスコア
	stCenterPoint						:TcVnVector2_DINT;									//ワークの中心座標格納用
	aGreen								:TcVnVector4_LREAL	:=[0, 255, 0, 0];				//緑色 (結果の描画用色)
	fbFormatString						:FB_FormatString;									//XY座標出力用
	
	//各実行時間を取得
	aPreprocessingDcTime				:ARRAY[0..1] OF T_DCTIME64;
	aInferenceDcTime					:ARRAY[0..1] OF T_DCTIME64;
	aPostprocessingDcTime				:ARRAY[0..1] OF T_DCTIME64;
	
	lrPreprocessingTime					:LREAL;
	lrInferenceTime						:LREAL;
	lrPostprocessingTime				:LREAL;
	

END_VAR

//---ONNXモデルのロード（起動時に1回だけ実行）---
	IF NOT bDnnModelInitialized THEN
		sFilePath := CONCAT(cFolderPath, cFileName);
		FW_SafeRelease(ADR(ipDnnModel)); //初期化前に念のためメモリ解放
		fbReadDnn(sFilePath := sFilePath, ipDestNeuralNetwork := ipDnnModel, bRead := TRUE, nTimeout:=T#10S);
		
		IF NOT fbReadDnn.bBusy THEN
			fbReadDnn(sFilePath:='', bRead := FALSE);
			IF NOT fbReadDnn.bError THEN
				bDnnModelInitialized := TRUE; //ロード大成功
			END_IF
			nReturnCode := fbReadDnn.nErrorId AND 16#FFF;
		END_IF
	END_IF


//---画像取得開始状態へ---
	eCameraState := F_VN_ApplicationSoftwareTrigger(fbCameraControl:=fbCameraControl);
	
	IF eCameraState <> TCVN_CS_ACQUIRING THEN
		RETURN;		//画像取込状態でなければ抜ける
	END_IF


//---画像取得後推論実施---
	CASE iStep OF
	0:
		fbR_TRIG(CLK := GVL.bAutoCameraTriger, Q => );
		
		IF fbR_TRIG.Q=TRUE THEN
			GVL.bLedLight:=TRUE;
		END_IF
	
		fbTon(IN:=GVL.bLedLight,PT:=T#500MS,Q=>,ET=>);	//LEDの照度安定待ち
		
		IF fbTon.Q=TRUE THEN
			bSoftWareTrigger:=TRUE;	//ソフトウェアトリガー
			iStep := 1;
		END_IF
		
	1:
		IF bSoftwareTrigger=TRUE THEN
			hr := fbCameraControl.TriggerImage();
			IF SUCCEEDED(hr)=TRUE THEN
				bSoftwareTrigger := FALSE;
			END_IF
		ELSE
			hr := fbCameraControl.GetCurrentImage(ipImageIn);	// 最新画像を取得			
			IF SUCCEEDED(hr)=TRUE AND ipImageIn <> 0 THEN
				GVL.bLedLight:=FALSE;
				iStep:=3;
			END_IF
		END_IF
		
	2:
		//NA
	
	3:
	//---プリプロセッシング---
	
		//DCタイムをゲット
		aPreprocessingDcTime[0]:=F_GetActualDcTime64();
		
		//1 BAYER_RGからRGBに変換
		hr := F_VN_ConvertColorSpace(ipImageIn, ipImageIn, TCVN_CST_BAYER_RG_TO_RGB, hr);
	
		//2 出力用画像に入力画像をコピー
		hr := F_VN_CopyImage(ipImageIn, ipimageOut, hr);
		
		//3 逆変換用の倍率とパディング（余白）を自動計算
		fScale:=MIN(UDINT_TO_REAL(cModelInputWidth)/cImageWidth, UDINT_TO_REAL(cModelInputHeight)/cImageHeight);		//アスペクト比を維持するため、縦横で縮小率のきつい方（小さい方）を基準倍率にする
		
		fPadX:=(UDINT_TO_REAL(cModelInputWidth)-(cImageWidth*fScale))/2.0;			//640x640 の中で、画像が中央配置されたときに発生する左右のグレー余白の幅を計算
		fPadY:=(UDINT_TO_REAL(cModelInputHeight)-(cImageHeight*fScale))/2.0;		//640x640 の中で、画像が中央配置されたときに発生する上下のグレー余白の幅を計算
		
		//4 ONNX入力に合わせて画像をリサイズ
		hr := F_VN_ResizeImageExp(ipImageIn, ipTensorImage, cModelInputWidth, cModelInputHeight, eInterpolationType, ePaddingMode, aGray, hr);
		
		//5 ONNX入力に合わせてfloat32(REAL)コンバート
		hr := F_VN_ConvertElementType(ipTensorImage, ipTensorImage, TCVN_ET_REAL, hr);
	
		//6 ONNX入力に合わせて4D Tensorの(バッチ, チャンネル, 縦, 横)に変換
		hr := F_VN_ConvertDataLayout(ipTensorImage, ipTensorImage, TCVN_DL_DEFAULT, TCVN_DL_4D_NCHW, hr);

		//DCタイムをゲット
		aPreprocessingDcTime[1]:=F_GetActualDcTime64();

		iStep:=4;
	
	4:
	//---ONNXに入力---
	
		//DCタイムをゲット
		aInferenceDcTime[0]:=F_GetActualDcTime64();
	
		hr := F_VN_ExecuteNeuralNetwork(ipDnnModel, ipTensorImage, ipDnnOutputImage, hr );
		
		//DCタイムをゲット
		aInferenceDcTime[1]:=F_GetActualDcTime64();
		
		iStep:=5;
		
	5:
	//---ポストプロセッシング---
	
		//DCタイムをゲット
		aPostprocessingDcTime[0]:=F_GetActualDcTime64();
	
		//0 コンテナ初期化
		hr := F_VN_CreateContainer(ipBoundingBoxes, ContainerType_Vector_TcVnRectangle_DINT, cNumBox, hr);		//NMS関数座標用
        hr := F_VN_CreateContainer(ipScores, ContainerType_Vector_REAL, cNumBox, hr);							//NMS関数スコア用
		
		hr := FW_SafeRelease(ADR(GVL.ipResultPoints));															//GVLにあるXY座標入力用コンテナをリリース(初回はコンテナ無いけど、大丈夫な関数)
		hr := F_VN_CreateContainer(GVL.ipResultPoints, ContainerType_Vector_TcVnPoint2_DINT, 0, hr);			//GVLにあるXY座標入力用コンテナ作成
		

        //1 ONNX実行結果の出力テンソル画像から、PLC上のREAL配列へコピー
        hr := F_VN_ExportImage(ipDnnOutputImage, ADR(aDnnRawOutput), SIZEOF(aDnnRawOutput), hr);
		
		//2 Row Dataを座標用コンテナに書き込み
		nIteratorIdx:=0;		//インデックスリセット
		hr := F_VN_GetForwardIterator(ipBoundingBoxes, ipIterator, hr);		//座標用コンテナから前方走査イテレータを取得
		IF SUCCEEDED(hr) AND ipIterator <> 0 THEN
			hr := ipIterator.TcQueryInterface(IID_ITcVnAccess_TcVnRectangle_DINT, ADR(ipAccessTcVnRectangleDINT));		//TcVnRectangle_DINT型アクセス用のアクセスインターフェースをクエリ
			IF SUCCEEDED(hr) AND ipAccessTcVnRectangleDINT <> 0 THEN
				WHILE SUCCEEDED(hr) AND ipIterator.CheckIfEnd() <> S_OK DO		//コンテナの終端に達するまで高速ループ
					
					stRectangle.nX			:=REAL_TO_DINT(aDnnRawOutput[0, nIteratorIdx, 0]-(aDnnRawOutput[0, nIteratorIdx, 2]/2.0));		// 計算式： 左上X ＝ 中心X － (幅 ÷ 2)
					stRectangle.nY			:=REAL_TO_DINT(aDnnRawOutput[0, nIteratorIdx, 1]-(aDnnRawOutput[0, nIteratorIdx, 3]/2.0));		// 計算式： 左上Y ＝ 中心Y － (高さ ÷ 2)
					stRectangle.nWidth		:=REAL_TO_DINT(aDnnRawOutput[0, nIteratorIdx, 2]);
					stRectangle.nHeight		:=REAL_TO_DINT(aDnnRawOutput[0, nIteratorIdx, 3]);		//YOLOXセンター座標（cx, cy）から、TwinCAT左上座標（x, y）に変換して中間バッファのストラクトに書き込み
				
					hr := ipAccessTcVnRectangleDINT.Set(stRectangle);		//アクセスインターフェース経由でデータをコンテナに書き込み
					
					IF SUCCEEDED(hr) THEN
						hr := ipIterator.Increment();
						nIteratorIdx:=nIteratorIdx+1;
					END_IF
					
				END_WHILE
			END_IF
			hr := FW_SafeRelease(ADR(ipAccessTcVnRectangleDINT));		//アクセスインターフェースを解放
		END_IF 
		hr := FW_SafeRelease(ADR(ipIterator));		//イテレータを解放


		//3 Row Dataをスコア用コンテナに書き込み
		nIteratorIdx:=0;		//インデックスリセット
		hr := F_VN_GetForwardIterator(ipScores, ipIterator, hr);		//スコア用コンテナから前方走査イテレータを取得
		IF SUCCEEDED(hr) AND ipIterator <> 0 THEN
			hr := ipIterator.TcQueryInterface(IID_ITcVnAccess_REAL, ADR(ipAccessREAL));		//REAL型アクセス用のアクセスインターフェースをクエリ
			IF SUCCEEDED(hr) AND ipAccessREAL <> 0 THEN
				WHILE SUCCEEDED(hr) AND ipIterator.CheckIfEnd() <> S_OK DO		//コンテナの終端に達するまで高速ループ
					
					hr := ipAccessREAL.Set(aDnnRawOutput[0, nIteratorIdx, 4] * aDnnRawOutput[0, nIteratorIdx, 5]);		//アクセスインターフェース経由でデータをコンテナに書き込み
																														//スコアはobj_score（物体らしさスコア）× class_score（クラススコア）					
					IF SUCCEEDED(hr) THEN
						hr := ipIterator.Increment();
						nIteratorIdx:=nIteratorIdx+1;
					END_IF
					
				END_WHILE
			END_IF
			hr := FW_SafeRelease(ADR(ipAccessREAL));		//アクセスインターフェースを解放
		END_IF 
		hr := FW_SafeRelease(ADR(ipIterator));		//イテレータを解放
		

		//4 Non-Maximum Suppression (NMS) の実行
        hr := F_VN_NonMaxSuppression(ipBoundingBoxes, ipScores, ipDestIndices, 0.3, 0.45, hr);		// 第4引数 (0.3)、第5引数（0.45）の説明コードの末尾にあり

		//NMS生存結果の抽出・描画・GVL出力
		hr := F_VN_GetNumberOfElements(ipDestIndices, nElementsFound, hr);		//NMSで生き残った（＝検出確定した）ワークの総数をカウント
		
		//1個以上ワークが検出された場合のみ、ループで1個ずつ処理を回す
		IF SUCCEEDED(hr) AND nElementsFound > 0 THEN
			
			FOR nIdx := 0 TO (ULINT_TO_UDINT(nElementsFound) - 1) DO
							
				hr := F_VN_GetAt_DINT(ipDestIndices, nTargetIndex, UDINT_TO_ULINT(nIdx), hr);		//NMSコンテナから、生き残った「元のRowDataのインデックス番号」を抽出

				hr := F_VN_GetAt_TcVnRectangle_DINT(ipBoundingBoxes, stFinalRect, DINT_TO_ULINT(nTargetIndex), hr);		//抽出したインデックスを使って、元の座標コンテナから長方形（Rect）データを取得
				
				hr := F_VN_GetAt_REAL(ipScores, fFinalScore, DINT_TO_ULINT(nTargetIndex), hr);		//抽出したインデックスを使って、元のスコアコンテナから確率データを取得

				// ONNXの座標から余白を引いて、縮小倍率で割り戻すことで、元画像のピクセル位置に戻す
				stFinalRect.nX      :=REAL_TO_DINT((DINT_TO_REAL(stFinalRect.nX) - fPadX) / fScale);
				stFinalRect.nY      :=REAL_TO_DINT((DINT_TO_REAL(stFinalRect.nY) - fPadY) / fScale);
				stFinalRect.nWidth  :=REAL_TO_DINT(DINT_TO_REAL(stFinalRect.nWidth) / fScale);
				stFinalRect.nHeight :=REAL_TO_DINT(DINT_TO_REAL(stFinalRect.nHeight) / fScale);
				
				//ワークの中心座標 (cx, cy) を計算し、DINT型構造体に落とし込む
				stCenterPoint[0]:=stFinalRect.nX + (stFinalRect.nWidth / 2);
				stCenterPoint[1]:=stFinalRect.nY + (stFinalRect.nHeight / 2);
				
				//確率表示にしたいので100倍
				fFinalScore:=fFinalScore*100.0;

				//ワーク幅から外れた物は無視
				IF (cWorkWidthMin<stFinalRect.nWidth AND stFinalRect.nWidth<cWorkWidthMax) AND (cWorkWidthMin<stFinalRect.nHeight AND stFinalRect.nHeight<cWorkWidthMax)  THEN
				
					//5 出力画像にワークの位置を画像に書き込み
					hr := F_VN_DrawRectangle(stFinalRect.nX, stFinalRect.nY, stFinalRect.nX+stFinalRect.nWidth, stFinalRect.nY + stFinalRect.nHeight,ipImageOut, aGreen, 2, hr);		//ワークを囲む長方形を描画
					
					hr := F_VN_DrawPoint(stCenterPoint[0], stCenterPoint[1], ipImageOut, TCVN_DS_PLUS, aGreen, hr);		//中心点に十字マークを描画
	
	
					//6 ワークのxy座標を画像に書き込み
					fbFormatString(	sFormat	:='( %2.1f ) = (%.3d, %.3d)', 
									arg1	:=F_REAL(fFinalScore),
									arg2	:=F_DINT(stCenterPoint[0]),
									arg3	:=F_DINT(stCenterPoint[1]));		//書き込み文字列生成
					
					hr := F_VN_PutText(fbFormatString.sOut, ipImageOut, stFinalRect.nX, stFinalRect.nY, TCVN_FT_HERSHEY_TRIPLEX, 0.5, aGreen, hr);		//XY座標を描画
					
					//7 GVLにあるコンテナにxy座標を書き込み
					hr := F_VN_AppendToContainer_TcVnVector2_DINT(stCenterPoint, GVL.ipResultPoints, hr);
		
				END_IF


			END_FOR
		END_IF
		
		//DCタイムをゲット
		aPostprocessingDcTime[1]:=F_GetActualDcTime64();
		
		iStep:=11;
		
	6..10:
		//NA

	11:
		//画面表示イメージを作成する
		hr := F_VN_TransformIntoDisplayableImage(ipImageIn, ipImageInDisp, hr);
        hr := F_VN_TransformIntoDisplayableImage(ipImageOut, ipImageOutDisp, hr);

		//ポインターの開放
		FW_SafeRelease(ADR(ipTensorImage));
		FW_SafeRelease(ADR(ipDnnOutputImage));
		FW_SafeRelease(ADR(ipBoundingBoxes));
		FW_SafeRelease(ADR(ipScores));
		FW_SafeRelease(ADR(ipDestIndices));
		
		//各実行時間を計算[ms]
		lrPreprocessingTime		:=ULINT_TO_LREAL(aPreprocessingDcTime[1]-aPreprocessingDcTime[0]) / 1000000.0;
		lrInferenceTime			:=ULINT_TO_LREAL(aInferenceDcTime[1]-aInferenceDcTime[0]) / 1000000.0;
		lrPostprocessingTime	:=ULINT_TO_LREAL(aPostprocessingDcTime[1]-aPostprocessingDcTime[0]) / 1000000.0;
		
        iStep := 0;
		
	END_CASE







(*ワンポイントメモ

NMS処理の引数説明
0.3 ＝ スコアの閾値（足切りライン）正式な引数名はfScoreThreshold
意味：
*直前で計算した「obj_score × class_score」の最終スコアが、「0.3（30%）未満のゴミ候補は、重なりを調べる前に最初から全部切り捨てる」という設定です。
現場での調整イメージ：
*誤検出（ワークがないのに背景を誤認識する）が多いとき			:この値を 0.4 や 0.5 に上げます。より自信のある候補しか残らなくなります。
*見落とし（あるはずのワークをスルーしてしまう）が多いとき		:この値を 0.2 や 0.15 に下げます。少し自信がなくても候補として拾うようになります。

2. 0.45 ＝ 重複の閾値（ダブり判定の基準）正式な引数名は fOverlapThreshold
意味：
*1つのワークに対して、AIが何個もダブって四角枠（ボックス）を出してしまったときに、「面積の45%以上が重なっていたら、それは同じワークを二重検出しているとみなして、スコアが低い方を消す」という設定です。
※この重なりの割合をAIの世界では「IoU（Intersection over Union）」と呼びます。
現場での調整イメージ：
*1つのワークに四角枠が2個も3個も重なって残ってしまうとき								:この値を 0.3 や 0.35 に下げます（重なりの判定を厳しくして、ちょっとでも重なっていたら容赦なく1個にまとめます）。
*ワーク同士が実際に近くに密集していて、隣のワークの枠まで巻き添えで消されてしまうとき	:この値を 0.55 や 0.6 に上げます（かなりガッツリ重なっていない限り、別々のワークとして認めるようになります）。

*)

END_PROGRAM

// ---- 04_Application/Vision/F_VN_ApplicationSoftwareTrigger.TcPOU
FUNCTION F_VN_ApplicationSoftwareTrigger	:ETcVnCameraState
VAR_INPUT
	fbCameraControl							:FB_VN_SimpleCameraControl;		// Cameraオブジェクト or File Sourceオブジェクト
END_VAR
VAR
	hr										:HRESULT;						// Vision関数の戻り値を表す変数
	eCameraState							:ETcVnCameraState;				// Cameraオブジェクト (or FileSourceオブジェクト) の状態を表す
END_VAR

// カメラのステータスを取得
eCameraState := fbCameraControl.GetState();

CASE eCameraState OF
TCVN_CS_ERROR:
	hr := fbCameraControl.Reset();					// エラーの時はリセットを実行

TCVN_CS_INITIAL..TCVN_CS_STARTACQUISITION:
	hr := fbCameraControl.StartAcquisition();		// 取込開始状態に移行させる

TCVN_CS_TRIGGERING:
	hr := fbCameraControl.TriggerImage();			// ソフトウェアトリガー
	
END_CASE

F_VN_ApplicationSoftwareTrigger := eCameraState;

END_FUNCTION

// ---- 04_Application/Vision/TcMlServer/P_MLSVision.TcPOU
PROGRAM P_MLSVision
VAR CONSTANT
	//カメラの画素数
	cImageWidth							:REAL	:=816.0;									//カメラ生画像の幅
    cImageHeight						:REAL	:=624.0;									//カメラ生画像の高さ
	
	//DNNモデルロード用
	cFolderPath							:STRING(255)	:='C:\TF7xxx_NeuralNetwork\';		//jsonファイルのディレクトリ
	cFileName							:STRING(255)	:='model_InDecode.json';			//jsonファイル名
	sMlSvrNetId							:T_AmsNetID		:='127.0.0.1.1.1';					//MLServer AMS Net ID
	eExecutionProvider					:E_EXECUTIONPROVIDER	:=E_EXECUTIONPROVIDER.CPU;	//CPU,CUDA使用選択
	
    //画像とモデルの解像度定義
    cModelInputWidth					:UDINT	:=640;										//ONNXモデルが要求する幅
    cModelInputHeight					:UDINT	:=640;										//ONNXモデルが要求する高さ

	//ONNXモデルリターン
	cBatchSize							:UDINT	:=1;										//バッチ数
    cNumBox								:UDINT	:=8400;										//ボックス数
    cElementPerBox						:UDINT	:=6;										//要素数	[cx, cy, w, h, obj_score, class_score]
	
	//ワーク幅
	cWorkWidthMin						:DINT	:=35;										//ワーク幅下限
	cWorkWidthMax						:DINT	:=50;										//ワーク幅上限
END_VAR
VAR
	//制御変数
	nIdx								:UDINT;												//ループ用
	iStep								:INT	:=0;										//画像処理のステップ進行用

	//カメラ・ライト制御
	bSoftWareTrigger					:BOOL;												//ソフトウェアトリガー
	fbR_TRIG							:R_TRIG;											//ボタンスイッチの立ち上がりエッジを検出
	fbTon								:ton;												//LEDライト点灯安定待ち

	//Vision必須関数
    hr									:HRESULT;											//Vision関数の戻り値を表す変数
    fbCameraControl						:FB_VN_SimpleCameraControl;							//Cameraオブジェクト or FileSourceオブジェクト
    eCameraState						:ETcVnCameraState;									//Cameraオブジェクト or FileSourceオブジェクト の状態
	
	//ポストプロセッシングで使用する倍率
	fScale								:REAL;												//レターボックスの縮小倍率
    fPadX								:REAL;												//X方向の余白（ピクセル）
    fPadY								:REAL;												//Y方向の余白（ピクセル）
	
	//model_InDecode用データ PlcOpenXmlより
	stModelInput						:ST_model_InDecodeInput;
	stModelOutput						:ST_model_InDecodeOutput;
	
	//マシンラーニングサーバー
	fbMlSvr								:FB_MlSvrPrediction();								//TcMlServerクライアントインスタンス
	sFilePath							:STRING(255);										//jsonファイルのファイルパス
	bMlSvrInitialized					:BOOL	:=FALSE;									//読み込み制御__________________________________後々はFB_Initにする
	bError								:BOOL;												//読み込みエラー
	
	//プリプロセッシング設定
	eInterpolationType					:ETcVnInterpolationType	:=TCVN_IT_BILINEAR;
	ePaddingMode						:ETcVnPaddingMode	:=TCVN_PM_LETTERBOX;
	aGray								:TcVnVector4_LREAL	:=[114, 114, 114, 0];			//グレー(レターボックス塗りつぶし色)
	
    //イメージ
    ipImageIn							:ITcVnImage;										//カメラからの生画像（816x624）
    ipTensorImage						:ITcVnImage;										//前処理（リサイズやREAL化）を施すテンソル
	ipImageOut							:ITcVnImage;										//結果の画像
	
	//表示用イメージ
	ipImageInDisp						:ITcVnDisplayableImage;								//入力画像の画面表示用変数
	ipImageOutDisp						:ITcVnDisplayableImage;								//結果画像の画面表示用変数

	//RowData書き込みコンテナ
	ipBoundingBoxes     				:ITcVnContainer;									//座標用コンテナ	(ContainerType_Vector_TcVnRectangle_DINT)
    ipScores            				:ITcVnContainer;									//スコア用コンテナ	(ContainerType_Vector_REAL)

    //コンテナアクセス用
    ipIterator							:ITcVnForwardIterator;								//イテレータ
    ipAccessTcVnRectangleDINT			:ITcVnAccess_TcVnRectangle_DINT;					//アクセスインターフェース(TcVnRectangle_DINT)
	ipAccessREAL						:ITcVnAccess_REAL;									//アクセスインターフェース(REAL)
	stRectangle							:TcVnRectangle_DINT;								//アクセスインターフェースに書き込む中間バッファ
	nIteratorIdx						:DINT;												//イテレータと一緒にカウント
	
	//NMS処理用
	ipDestIndices						:ITcVnContainer;									//NMSで残ったインデックス番号用コンテナ	(ContainerType_Vector_DINT)
	nElementsFound						:ULINT;												//NMSで生き残った確定ワーク数
	
	//結果の出力用
	nTargetIndex						:DINT;												//NMSで生き残った元のインデックス番号
	stFinalRect							:TcVnRectangle_DINT;								//最終確定したワークの座標
	fFinalScore							:REAL;												//最終確定したワークのスコア
	stCenterPoint						:TcVnVector2_DINT;									//ワークの中心座標格納用
	aGreen								:TcVnVector4_LREAL	:=[0, 255, 0, 0];				//緑色 (結果の描画用色)
	fbFormatString						:FB_FormatString;									//XY座標出力用
	
	//各実行時間を取得
	aPreprocessingDcTime				:ARRAY[0..1] OF T_DCTIME64;
	aInferenceDcTime					:ARRAY[0..1] OF T_DCTIME64;
	aPostprocessingDcTime				:ARRAY[0..1] OF T_DCTIME64;
	
	lrPreprocessingTime					:LREAL;
	lrInferenceTime						:LREAL;
	lrPostprocessingTime				:LREAL;
	


END_VAR

//---MLServerクライアントのインスタンス化---
	IF NOT bMlSvrInitialized THEN
		sFilePath := CONCAT(cFolderPath, cFileName);
		
		//サーバー設定をFBに入力
		fbMlSvr.stPredictionParameter.sMlModelFilePath		:=sFilePath;
		fbMlSvr.stPredictionParameter.sMlSvrNetId			:=sMlSvrNetId;
		fbMlSVr.stPredictionParameter.eExecutionProvider	:=eExecutionProvider;  
		
		IF fbMlSvr.Configure(nTimeout := 1000, nPriority:=0) THEN
			IF fbMlSvr.nErrorCode <> 0 THEN
				bError:=TRUE;
			ELSE
				bMlSvrInitialized := TRUE; //ロード大成功
			END_IF
		END_IF
		
		
	END_IF




//---画像取得開始状態へ---
	eCameraState := F_VN_ApplicationSoftwareTrigger(fbCameraControl:=fbCameraControl);
	
	IF eCameraState <> TCVN_CS_ACQUIRING THEN
		RETURN;		//画像取込状態でなければ抜ける
	END_IF


//---画像取得後推論実施---
	CASE iStep OF
	0:
		fbR_TRIG(CLK := GVL.bAutoCameraTriger, Q => );
		
		IF fbR_TRIG.Q=TRUE THEN
			GVL.bLedLight:=TRUE;
		END_IF
	
		fbTon(IN:=GVL.bLedLight,PT:=T#500MS,Q=>,ET=>);	//LEDの照度安定待ち
		
		IF fbTon.Q=TRUE THEN
			bSoftWareTrigger:=TRUE;	//ソフトウェアトリガー
			iStep := 1;
		END_IF
		
	1:
		IF bSoftwareTrigger=TRUE THEN
			hr := fbCameraControl.TriggerImage();
			IF SUCCEEDED(hr)=TRUE THEN
				bSoftwareTrigger := FALSE;
			END_IF
		ELSE
			hr := fbCameraControl.GetCurrentImage(ipImageIn);	// 最新画像を取得			
			IF SUCCEEDED(hr)=TRUE AND ipImageIn <> 0 THEN
				GVL.bLedLight:=FALSE;
				iStep:=3;
			END_IF
		END_IF
		
	2:
		//NA
	
	3:
	//---プリプロセッシング---
	
		//DCタイムをゲット
		aPreprocessingDcTime[0]:=F_GetActualDcTime64();
		
		//1 BAYER_RGからRGBに変換
		hr := F_VN_ConvertColorSpace(ipImageIn, ipImageIn, TCVN_CST_BAYER_RG_TO_RGB, hr);
	
		//2 出力用画像に入力画像をコピー
		hr := F_VN_CopyImage(ipImageIn, ipimageOut, hr);
		
		//3 逆変換用の倍率とパディング（余白）を自動計算
		fScale:=MIN(UDINT_TO_REAL(cModelInputWidth)/cImageWidth, UDINT_TO_REAL(cModelInputHeight)/cImageHeight);		//アスペクト比を維持するため、縦横で縮小率のきつい方（小さい方）を基準倍率にする
		
		fPadX:=(UDINT_TO_REAL(cModelInputWidth)-(cImageWidth*fScale))/2.0;			//640x640 の中で、画像が中央配置されたときに発生する左右のグレー余白の幅を計算
		fPadY:=(UDINT_TO_REAL(cModelInputHeight)-(cImageHeight*fScale))/2.0;		//640x640 の中で、画像が中央配置されたときに発生する上下のグレー余白の幅を計算
		
		//4 ONNX入力に合わせて画像をリサイズ
		hr := F_VN_ResizeImageExp(ipImageIn, ipTensorImage, cModelInputWidth, cModelInputHeight, eInterpolationType, ePaddingMode, aGray, hr);
		
		//5 ONNX入力に合わせてfloat32(REAL)コンバート
		hr := F_VN_ConvertElementType(ipTensorImage, ipTensorImage, TCVN_ET_REAL, hr);
	
		//6 ONNX入力に合わせて4D Tensorの(バッチ, チャンネル, 縦, 横)に変換
		hr := F_VN_ConvertDataLayout(ipTensorImage, ipTensorImage, TCVN_DL_DEFAULT, TCVN_DL_4D_NCHW, hr);
		
		//7 Tensor画像をPLC上のREAL配列へコピー
        hr := F_VN_ExportImage(ipTensorImage, ADR(stModelInput.in_images), SIZEOF(stModelInput.in_images), hr);

		//DCタイムをゲット
		aPreprocessingDcTime[1]:=F_GetActualDcTime64();

		iStep:=4;
	
	4:
	//---推論実行---
	
		//DCタイムをゲット
		aInferenceDcTime[0]:=F_GetActualDcTime64();
	
		IF bMlSvrInitialized AND NOT bError THEN
			IF fbMlSvr.Predict(	pDataIn			:= ADR(stModelInput), 
								nDataInSize		:= SIZEOF(stModelInput), 
								pDataOut		:= ADR(stModelOutput), 
								nDataOutSize	:= SIZEOF(stModelOutput),
								nTimeout		:= 1000,
								nPriority		:= 0) THEN
								
				IF fbMlSvr.nErrorCode <> 0 THEN
					bError := TRUE;
				ELSE
					//DCタイムをゲット
					aInferenceDcTime[1]:=F_GetActualDcTime64();
					
					iStep:=5;
				END_IF
				
			END_IF
		END_IF
		
		
	5:
	//---ポストプロセッシング---
	
